C09102=1029.848,308.460,372.432,171.179,46.085,158.925
C09103=1029.841,308.212,372.466,171.174,46.085,158.924
C09104=1029.833,307.965,372.499,171.169,46.086,158.924
C09105=1029.826,307.717,372.532,171.165,46.085,158.923
C09106=1029.819,307.470,372.565,171.160,46.086,158.923
C09107=1029.807,307.057,372.620,171.152,46.086,158.922
C09108=1029.795,306.645,372.676,171.145,46.086,158.921
C09109=1029.784,306.233,372.731,171.136,46.086,158.920
C09110=1029.772,305.821,372.786,171.128,46.087,158.919
C09111=1029.765,305.573,372.819,171.124,46.087,158.919
C09112=1029.758,305.326,372.853,171.119,46.087,158.918
C09113=1029.751,305.077,372.886,171.115,46.087,158.918
C09114=1029.744,304.831,372.919,171.110,46.087,158.917
C09115=1029.737,304.582,372.952,171.105,46.088,158.917
C09116=1029.731,304.335,372.985,171.100,46.088,158.916
C09117=1029.723,304.087,373.018,171.096,46.088,158.916
C09118=1029.717,303.840,373.051,171.092,46.088,158.915
C09119=1029.709,303.592,373.085,171.087,46.088,158.915
C09120=1029.703,303.344,373.117,171.082,46.089,158.914
C09121=1029.695,303.097,373.150,171.077,46.088,158.914
C09122=1029.689,302.850,373.183,171.073,46.089,158.913
C09123=1029.682,302.601,373.216,171.069,46.089,158.913
C09124=1029.674,302.353,373.249,171.064,46.089,158.912
C09125=1029.668,302.106,373.282,171.060,46.089,158.912
C09126=1029.661,301.859,373.315,171.054,46.090,158.911
C09127=1029.654,301.610,373.348,171.050,46.090,158.911
C09128=1029.647,301.363,373.380,171.045,46.090,158.911
C09129=1029.641,301.115,373.413,171.041,46.090,158.910
C09130=1029.634,300.867,373.446,171.037,46.091,158.910
C09131=1029.626,300.620,373.479,171.033,46.091,158.909
C09132=1029.620,300.372,373.512,171.028,46.091,158.909
C09133=1029.613,300.124,373.545,171.023,46.092,158.908
C09134=1029.606,299.877,373.577,171.018,46.092,158.908
C09135=1029.600,299.629,373.610,171.014,46.092,158.907
C09136=1029.593,299.381,373.643,171.009,46.092,158.907
C09137=1029.586,299.134,373.675,171.005,46.093,158.906
C09138=1029.579,298.885,373.708,171.001,46.093,158.906
C09139=1029.573,298.638,373.741,170.996,46.093,158.906
C09140=1029.566,298.390,373.774,170.992,46.094,158.905
C09141=1029.559,298.142,373.806,170.988,46.094,158.905
C09142=1029.552,297.894,373.839,170.983,46.094,158.904
C09143=1029.546,297.647,373.872,170.978,46.094,158.904
C09144=1029.539,297.399,373.904,170.973,46.095,158.903
C09145=1029.532,297.151,373.937,170.969,46.095,158.903
C09146=1029.526,296.904,373.970,170.965,46.096,158.903
C09147=1029.518,296.656,374.002,170.961,46.096,158.902
C09148=1029.512,296.408,374.035,170.956,46.096,158.902
C09149=1029.506,296.161,374.068,170.952,46.097,158.901
C09150=1029.499,295.913,374.100,170.948,46.097,158.901
C09151=1029.492,295.665,374.133,170.943,46.097,158.900
C09152=1029.486,295.417,374.166,170.939,46.097,158.900
C09153=1029.479,295.169,374.197,170.934,46.098,158.900
C09154=1029.473,294.922,374.230,170.930,46.098,158.899
C09155=1029.466,294.674,374.263,170.926,46.098,158.899
C09156=1029.459,294.426,374.295,170.921,46.099,158.898
C09157=1029.452,294.179,374.328,170.917,46.099,158.898
C09158=1029.446,293.931,374.360,170.913,46.099,158.897
C09159=1029.439,293.684,374.392,170.909,46.100,158.897
C09160=1029.432,293.435,374.425,170.904,46.101,158.897
C09161=1029.425,293.187,374.456,170.900,46.101,158.896
C09162=1029.418,292.940,374.488,170.895,46.102,158.896
C09163=1029.407,292.544,374.540,170.888,46.103,158.895
C09164=1029.397,292.150,374.591,170.882,46.103,158.895
C09165=1029.385,291.754,374.642,170.874,46.104,158.894
C09166=1029.375,291.359,374.693,170.868,46.105,158.894
C09167=1029.368,291.112,374.725,170.864,46.105,158.893
C09168=1029.361,290.864,374.757,170.860,46.106,158.893
C09169=1029.354,290.616,374.788,170.854,46.107,158.893
C09170=1029.348,290.367,374.821,170.850,46.107,158.892
C09171=1029.341,290.120,374.853,170.846,46.108,158.892
C09172=1029.334,289.872,374.884,170.842,46.109,158.891
C09173=1029.327,289.625,374.916,170.837,46.109,158.891
C09174=1029.320,289.377,374.948,170.833,46.109,158.891
C09175=1029.314,289.129,374.980,170.829,46.110,158.890
C09176=1029.307,288.882,375.012,170.825,46.111,158.890
C09177=1029.300,288.633,375.044,170.820,46.111,158.890
C09178=1029.293,288.385,375.075,170.816,46.112,158.889
C09179=1029.286,288.137,375.107,170.812,46.113,158.889
C09180=1029.279,287.890,375.139,170.808,46.113,158.889
C09181=1029.273,287.642,375.170,170.804,46.114,158.888
C09182=1029.267,287.394,375.202,170.799,46.114,158.888
C09183=1029.260,287.146,375.234,170.795,46.115,158.888
C09184=1029.253,286.899,375.266,170.791,46.116,158.887
C09185=1029.246,286.651,375.297,170.787,46.117,158.887
C09186=1029.239,286.403,375.329,170.783,46.117,158.887
C09187=1029.233,286.155,375.360,170.778,46.117,158.886
C09188=1029.226,285.907,375.392,170.774,46.118,158.886
C09189=1029.219,285.658,375.423,170.770,46.119,158.886
C09190=1029.212,285.410,375.455,170.766,46.120,158.885
C09191=1029.205,285.163,375.486,170.762,46.121,158.885
C09192=1029.198,284.915,375.518,170.757,46.121,158.885
C09193=1029.192,284.667,375.549,170.753,46.122,158.884
C09194=1029.185,284.419,375.581,170.749,46.123,158.884
C09195=1029.178,284.171,375.612,170.745,46.124,158.884
C09196=1029.172,283.923,375.643,170.741,46.124,158.883
C09197=1029.164,283.675,375.674,170.737,46.125,158.883
C09198=1029.157,283.428,375.706,170.733,46.126,158.883
C09199=1029.151,283.180,375.737,170.729,46.126,158.883
C09200=1029.144,282.932,375.769,170.725,46.127,158.882
C09201=1029.137,282.684,375.800,170.721,46.128,158.882
C09202=1029.130,282.436,375.831,170.717,46.128,158.882
C09203=1029.124,282.187,375.862,170.713,46.129,158.881
C09204=1029.117,281.939,375.894,170.709,46.130,158.881
C09205=1029.111,281.692,375.925,170.705,46.131,158.881
C09206=1029.103,281.444,375.956,170.701,46.132,158.881
C09207=1029.097,281.197,375.987,170.696,46.133,158.880
C09208=1029.091,280.948,376.018,170.692,46.133,158.880
C09209=1029.084,280.700,376.049,170.688,46.134,158.880
C09210=1029.077,280.452,376.080,170.684,46.135,158.879
C09211=1029.070,280.205,376.112,170.680,46.136,158.879
C09212=1029.064,279.956,376.143,170.676,46.137,158.879
C09213=1029.057,279.708,376.174,170.672,46.138,158.879
C09214=1029.051,279.460,376.205,170.668,46.139,158.878
C09215=1029.043,279.213,376.236,170.664,46.139,158.878
C09216=1029.037,278.965,376.267,170.660,46.140,158.878
C09217=1029.031,278.717,376.298,170.656,46.141,158.877
C09218=1029.024,278.469,376.330,170.652,46.142,158.877
C09219=1029.014,278.086,376.377,170.646,46.143,158.877
C09220=1029.003,277.703,376.426,170.640,46.144,158.876
C09221=1028.993,277.320,376.473,170.634,46.146,158.876
C09222=1028.983,276.937,376.521,170.628,46.147,158.876
C09223=1028.976,276.689,376.551,170.624,46.148,158.875
C09224=1028.969,276.441,376.582,170.619,46.149,158.875
C09225=1028.963,276.193,376.612,170.615,46.150,158.875
C09226=1028.956,275.946,376.643,170.611,46.151,158.874
C09227=1028.949,275.697,376.674,170.607,46.152,158.874
C09228=1028.942,275.449,376.705,170.603,46.153,158.874
C09229=1028.935,275.201,376.736,170.599,46.154,158.874
C09230=1028.930,274.953,376.766,170.596,46.154,158.874
C09231=1028.923,274.705,376.797,170.592,46.155,158.873
C09232=1028.916,274.457,376.827,170.588,46.156,158.873
C09233=1028.909,274.209,376.859,170.584,46.157,158.873
C09234=1028.902,273.962,376.889,170.580,46.158,158.873
C09235=1028.896,273.713,376.919,170.576,46.159,158.872
C09236=1028.889,273.465,376.951,170.572,46.160,158.872
C09237=1028.882,273.217,376.981,170.568,46.161,158.872
C09238=1028.876,272.969,377.011,170.564,46.162,158.872
C09239=1028.869,272.721,377.041,170.561,46.163,158.871
C09240=1028.862,272.473,377.073,170.557,46.164,158.871
C09241=1028.855,272.225,377.103,170.553,46.165,158.871
C09242=1028.849,271.977,377.133,170.549,46.166,158.871
C09243=1028.842,271.729,377.163,170.545,46.167,158.870
C09244=1028.836,271.480,377.194,170.540,46.168,158.870
C09245=1028.829,271.233,377.225,170.537,46.170,158.870
C09246=1028.823,270.985,377.255,170.534,46.170,158.870
C09247=1028.816,270.736,377.286,170.530,46.172,158.870
C09248=1028.810,270.489,377.316,170.526,46.173,158.870
C09249=1028.803,270.240,377.347,170.522,46.174,158.869
C09250=1028.796,269.992,377.377,170.518,46.175,158.869
C09251=1028.789,269.744,377.406,170.513,46.176,158.869
C09252=1028.783,269.496,377.437,170.511,46.177,158.869
C09253=1028.776,269.248,377.467,170.507,46.178,158.869
C09254=1028.769,269.000,377.497,170.503,46.179,158.868
C09255=1028.763,268.752,377.528,170.499,46.180,158.868
C09256=1028.756,268.504,377.558,170.495,46.181,158.868
C09257=1028.750,268.256,377.588,170.491,46.183,158.868
C09258=1028.743,268.007,377.618,170.487,46.184,158.867
C09259=1028.736,267.760,377.648,170.484,46.184,158.867
C09260=1028.730,267.511,377.679,170.480,46.185,158.867
C09261=1028.723,267.263,377.709,170.476,46.187,158.867
C09262=1028.716,267.016,377.739,170.472,46.188,158.867
C09263=1028.710,266.767,377.769,170.468,46.189,158.867
C09264=1028.703,266.520,377.799,170.465,46.190,158.867
C09265=1028.696,266.271,377.829,170.461,46.191,158.866
C09266=1028.689,266.023,377.860,170.457,46.192,158.866
C09267=1028.683,265.775,377.889,170.453,46.194,158.866
C09268=1028.676,265.527,377.919,170.449,46.195,158.866
C09269=1028.670,265.279,377.949,170.445,46.196,158.865
C09270=1028.662,265.031,377.979,170.442,46.197,158.865
C09271=1028.657,264.782,378.009,170.438,46.198,158.865
C09272=1028.650,264.534,378.039,170.434,46.199,158.865
C09273=1028.643,264.286,378.069,170.431,46.201,158.865
C09274=1028.636,264.039,378.099,170.427,46.202,158.865
C09275=1028.626,263.660,378.144,170.422,46.204,158.865
C09276=1028.616,263.282,378.189,170.416,46.205,158.864
C09277=1028.606,262.904,378.235,170.410,46.208,158.864
C09278=1028.595,262.525,378.280,170.404,46.210,158.864
C09279=1028.590,262.277,378.311,170.400,46.211,158.864
C09280=1028.583,262.029,378.340,170.397,46.212,158.864
C09281=1028.576,261.781,378.370,170.393,46.213,158.863
C09282=1028.569,261.532,378.399,170.390,46.215,158.863
C09283=1028.563,261.285,378.429,170.385,46.216,158.863
C09284=1028.557,261.037,378.460,170.382,46.217,158.863
C09285=1028.549,260.788,378.488,170.379,46.218,158.863
C09286=1028.543,260.541,378.518,170.375,46.220,158.863
C09287=1028.536,260.292,378.547,170.371,46.221,158.862
C09288=1028.530,260.044,378.577,170.367,46.223,158.862
C09289=1028.523,259.796,378.607,170.363,46.224,158.862
C09290=1028.516,259.548,378.635,170.360,46.225,158.862
C09291=1028.509,259.299,378.665,170.357,46.227,158.862
C09292=1028.502,259.052,378.694,170.353,46.228,158.862
C09293=1028.495,258.803,378.724,170.349,46.229,158.862
C09294=1028.489,258.555,378.753,170.345,46.231,158.862
C09295=1028.481,258.307,378.782,170.341,46.233,158.861
C09296=1028.475,258.059,378.811,170.339,46.234,158.861
C09297=1028.468,257.810,378.841,170.334,46.235,158.861
C09298=1028.462,257.562,378.870,170.331,46.237,158.861
C09299=1028.455,257.314,378.899,170.327,46.238,158.861
C09300=1028.448,257.066,378.928,170.323,46.239,158.861
C09301=1028.441,256.817,378.957,170.320,46.241,158.861
C09302=1028.434,256.569,378.987,170.316,46.242,158.861
C09303=1028.428,256.321,379.016,170.313,46.244,158.861
C09304=1028.422,256.073,379.046,170.309,46.245,158.860
C09305=1028.414,255.824,379.074,170.306,46.246,158.860
C09306=1028.408,255.576,379.103,170.302,46.248,158.860
C09307=1028.401,255.328,379.134,170.298,46.250,158.860
C09308=1028.395,255.080,379.163,170.294,46.251,158.860
C09309=1028.388,254.832,379.191,170.291,46.252,158.860
C09310=1028.381,254.583,379.220,170.288,46.254,158.860
C09311=1028.375,254.335,379.249,170.284,46.255,158.860
C09312=1028.368,254.087,379.278,170.280,46.257,158.860
C09313=1028.361,253.838,379.308,170.276,46.258,158.860
C09314=1028.354,253.591,379.337,170.273,46.259,158.860
C09315=1028.348,253.343,379.366,170.270,46.261,158.859
C09316=1028.341,253.094,379.395,170.266,46.263,158.859
C09317=1028.335,252.846,379.425,170.262,46.264,158.859
C09318=1028.328,252.598,379.453,170.259,46.266,158.859
C09319=1028.322,252.350,379.482,170.255,46.267,158.859
C09320=1028.315,252.101,379.511,170.252,46.268,158.859
C09321=1028.308,251.853,379.540,170.249,46.270,158.859
C09322=1028.302,251.605,379.570,170.245,46.271,158.859
C09323=1028.295,251.356,379.598,170.241,46.273,158.859
C09324=1028.288,251.108,379.627,170.238,46.275,158.859
C09325=1028.282,250.860,379.656,170.235,46.275,158.859
C09326=1028.276,250.612,379.685,170.231,46.277,158.858
C09327=1028.269,250.364,379.714,170.227,46.279,158.858
C09328=1028.262,250.115,379.743,170.224,46.280,158.858
C09329=1028.256,249.867,379.772,170.221,46.282,158.858
C09330=1028.250,249.619,379.801,170.217,46.283,158.858
C09331=1028.239,249.239,379.846,170.211,46.286,158.858
C09332=1028.229,248.860,379.890,170.206,46.288,158.858
C09333=1028.220,248.480,379.933,170.201,46.290,158.858
C09334=1028.210,248.100,379.978,170.196,46.292,158.858
C09335=1028.203,247.852,380.007,170.192,46.294,158.858
C09336=1028.196,247.604,380.035,170.188,46.296,158.858
C09337=1028.190,247.356,380.064,170.186,46.297,158.858
C09338=1028.184,247.107,380.093,170.182,46.299,158.857
C09339=1028.178,246.859,380.122,170.178,46.300,158.857
C09340=1028.170,246.610,380.150,170.175,46.302,158.857
C09341=1028.164,246.362,380.179,170.172,46.303,158.857
C09342=1028.158,246.114,380.208,170.168,46.305,158.857
C09343=1028.151,245.866,380.237,170.165,46.306,158.857
C09344=1028.145,245.617,380.265,170.161,46.308,158.857
C09345=1028.139,245.369,380.294,170.158,46.310,158.857
C09346=1028.132,245.121,380.323,170.155,46.311,158.857
C09347=1028.126,244.873,380.352,170.151,46.313,158.857
C09348=1028.119,244.624,380.380,170.147,46.314,158.857
C09349=1028.113,244.376,380.409,170.145,46.316,158.857
C09350=1028.106,244.128,380.438,170.141,46.317,158.857
C09351=1028.100,243.879,380.466,170.137,46.319,158.857
C09352=1028.093,243.631,380.495,170.134,46.320,158.857
C09353=1028.087,243.383,380.523,170.131,46.322,158.857
C09354=1028.080,243.134,380.552,170.127,46.324,158.856
C09355=1028.073,242.887,380.580,170.124,46.326,158.857
C09356=1028.067,242.638,380.609,170.121,46.327,158.857
C09357=1028.061,242.390,380.637,170.117,46.329,158.856
C09358=1028.055,242.141,380.666,170.114,46.331,158.856
C09359=1028.048,241.893,380.694,170.110,46.332,158.856
C09360=1028.042,241.645,380.722,170.107,46.334,158.856
C09361=1028.035,241.397,380.751,170.104,46.336,158.856
C09362=1028.029,241.148,380.779,170.100,46.338,158.856
C09363=1028.022,240.900,380.808,170.097,46.339,158.856
C09364=1028.014,240.651,380.836,170.094,46.341,158.856
C09365=1028.008,240.403,380.865,170.090,46.342,158.856
C09366=1028.002,240.155,380.892,170.086,46.344,158.856
C09367=1027.996,239.906,380.921,170.084,46.346,158.856
C09368=1027.989,239.658,380.949,170.080,46.348,158.856
C09369=1027.982,239.410,380.977,170.076,46.349,158.856
C09370=1027.975,239.161,381.005,170.074,46.351,158.856
C09371=1027.969,238.913,381.034,170.070,46.353,158.856
C09372=1027.962,238.665,381.061,170.066,46.355,158.856
C09373=1027.956,238.416,381.089,170.064,46.357,158.856
C09374=1027.949,238.168,381.117,170.060,46.358,158.856
C09375=1027.942,237.920,381.145,170.056,46.360,158.856
C09376=1027.936,237.671,381.174,170.054,46.362,158.856
C09377=1027.929,237.423,381.201,170.050,46.364,158.856
C09378=1027.923,237.174,381.229,170.046,46.365,158.856
C09379=1027.916,236.926,381.258,170.044,46.367,158.856
C09380=1027.909,236.678,381.285,170.040,46.369,158.856
C09381=1027.903,236.429,381.314,170.037,46.371,158.856
C09382=1027.896,236.181,381.341,170.034,46.373,158.856
C09383=1027.890,235.932,381.369,170.030,46.374,158.856
C09384=1027.883,235.684,381.397,170.027,46.377,158.856
C09385=1027.877,235.437,381.425,170.024,46.378,158.856
C09386=1027.870,235.188,381.453,170.020,46.380,158.856
C09387=1027.859,234.802,381.496,170.015,46.383,158.856
C09388=1027.850,234.417,381.539,170.010,46.386,158.856
C09389=1027.839,234.031,381.582,170.005,46.389,158.856
C09390=1027.829,233.645,381.626,170.000,46.392,158.856
C09391=1027.823,233.397,381.653,169.997,46.394,158.856
C09392=1027.816,233.148,381.681,169.993,46.395,158.856
C09393=1027.810,232.900,381.709,169.991,46.397,158.856
C09394=1027.803,232.651,381.737,169.987,46.399,158.856
C09395=1027.797,232.403,381.765,169.983,46.401,158.856
C09396=1027.790,232.154,381.792,169.981,46.403,158.856
C09397=1027.783,231.906,381.820,169.977,46.405,158.857
C09398=1027.777,231.657,381.848,169.973,46.407,158.856
C09399=1027.770,231.410,381.875,169.971,46.409,158.857
C09400=1027.764,231.161,381.903,169.967,46.410,158.856
C09401=1027.758,230.913,381.931,169.965,46.412,158.857
C09402=1027.751,230.664,381.959,169.961,46.414,158.857
C09403=1027.744,230.416,381.987,169.958,46.416,158.857
C09404=1027.738,230.167,382.015,169.955,46.418,158.857
C09405=1027.731,229.918,382.041,169.951,46.420,158.857
C09406=1027.725,229.671,382.068,169.948,46.422,158.857
C09407=1027.718,229.422,382.096,169.945,46.424,158.857
C09408=1027.711,229.174,382.124,169.942,46.426,158.857
C09409=1027.705,228.925,382.152,169.939,46.427,158.857
C09410=1027.698,228.677,382.179,169.935,46.430,158.857
C09411=1027.691,228.428,382.206,169.932,46.432,158.857
C09412=1027.685,228.180,382.234,169.929,46.434,158.857
C09413=1027.679,227.932,382.261,169.926,46.436,158.857
C09414=1027.672,227.683,382.289,169.923,46.438,158.857
C09415=1027.665,227.435,382.317,169.920,46.440,158.857
C09416=1027.660,227.186,382.343,169.916,46.442,158.857
C09417=1027.653,226.938,382.371,169.914,46.444,158.857
C09418=1027.645,226.690,382.398,169.910,46.446,158.857
C09419=1027.639,226.441,382.425,169.906,46.448,158.857
C09420=1027.632,226.192,382.453,169.904,46.450,158.858
C09421=1027.626,225.945,382.480,169.900,46.452,158.858
C09422=1027.619,225.696,382.507,169.898,46.454,158.858
C09423=1027.613,225.447,382.535,169.894,46.456,158.858
C09424=1027.606,225.198,382.562,169.891,46.458,158.858
C09425=1027.600,224.950,382.589,169.888,46.460,158.858
C09426=1027.593,224.703,382.616,169.884,46.462,158.858
C09427=1027.586,224.453,382.643,169.881,46.464,158.858
C09428=1027.580,224.205,382.671,169.879,46.466,158.858
C09429=1027.573,223.956,382.697,169.875,46.469,158.858
C09430=1027.566,223.709,382.725,169.873,46.471,158.858
C09431=1027.560,223.459,382.752,169.869,46.472,158.858
C09432=1027.553,223.211,382.779,169.865,46.475,158.858
C09433=1027.546,222.963,382.807,169.863,46.477,158.858
C09434=1027.540,222.715,382.833,169.859,46.479,158.859
C09435=1027.534,222.466,382.861,169.857,46.481,158.859
C09436=1027.527,222.217,382.888,169.853,46.483,158.859
C09437=1027.520,221.970,382.915,169.850,46.485,158.859
C09438=1027.514,221.721,382.942,169.847,46.487,158.859
C09439=1027.507,221.472,382.969,169.844,46.490,158.859
C09440=1027.501,221.224,382.995,169.841,46.492,158.859
C09441=1027.494,220.975,383.023,169.838,46.493,158.859
C09442=1027.488,220.727,383.050,169.834,46.496,158.859
C09443=1027.477,220.333,383.093,169.830,46.499,158.859
C09444=1027.467,219.940,383.136,169.825,46.502,158.859
C09445=1027.456,219.546,383.179,169.819,46.506,158.859
C09446=1027.447,219.153,383.221,169.815,46.509,158.860
C09447=1027.440,218.904,383.248,169.812,46.511,158.860
C09448=1027.433,218.656,383.275,169.809,46.513,158.860
C09449=1027.427,218.407,383.301,169.806,46.516,158.860
C09450=1027.420,218.159,383.329,169.802,46.518,158.860
C09451=1027.413,217.910,383.355,169.800,46.520,158.860
C09452=1027.407,217.662,383.382,169.796,46.522,158.860
C09453=1027.400,217.413,383.408,169.794,46.524,158.860
C09454=1027.393,217.164,383.435,169.791,46.527,158.861
C09455=1027.387,216.917,383.462,169.787,46.529,158.861
C09456=1027.380,216.668,383.489,169.785,46.531,158.861
C09457=1027.374,216.420,383.515,169.781,46.534,158.861
C09458=1027.367,216.171,383.541,169.779,46.536,158.861
C09459=1027.360,215.922,383.568,169.775,46.538,158.861
C09460=1027.353,215.675,383.595,169.772,46.540,158.861
C09461=1027.347,215.425,383.622,169.769,46.542,158.861
C09462=1027.341,215.177,383.648,169.766,46.545,158.861
C09463=1027.334,214.928,383.675,169.763,46.547,158.862
C09464=1027.327,214.680,383.702,169.760,46.549,158.862
C09465=1027.321,214.432,383.728,169.756,46.551,158.862
C09466=1027.314,214.182,383.755,169.754,46.554,158.862
C09467=1027.308,213.934,383.781,169.751,46.556,158.862
C09468=1027.301,213.686,383.808,169.748,46.558,158.862
C09469=1027.294,213.438,383.834,169.745,46.561,158.862
C09470=1027.288,213.189,383.861,169.742,46.563,158.862
C09471=1027.281,212.940,383.888,169.739,46.565,158.863
C09472=1027.274,212.692,383.914,169.735,46.567,158.863
C09473=1027.268,212.443,383.941,169.733,46.570,158.863
C09474=1027.262,212.195,383.967,169.730,46.572,158.863
C09475=1027.255,211.946,383.994,169.727,46.574,158.863
C09476=1027.249,211.698,384.020,169.724,46.576,158.863
C09477=1027.242,211.449,384.047,169.721,46.578,158.863
C09478=1027.236,211.201,384.073,169.718,46.581,158.863
C09479=1027.229,210.952,384.100,169.715,46.583,158.864
C09480=1027.223,210.704,384.126,169.712,46.586,158.864
C09481=1027.216,210.455,384.153,169.709,46.588,158.864
C09482=1027.209,210.207,384.179,169.706,46.590,158.864
C09483=1027.202,209.958,384.205,169.703,46.592,158.864
C09484=1027.196,209.710,384.232,169.700,46.595,158.864
C09485=1027.189,209.461,384.258,169.697,46.598,158.864
C09486=1027.183,209.213,384.284,169.695,46.600,158.865
C09487=1027.176,208.964,384.310,169.691,46.602,158.865
C09488=1027.170,208.715,384.337,169.689,46.605,158.865
C09489=1027.164,208.467,384.363,169.685,46.607,158.865
C09490=1027.157,208.218,384.389,169.682,46.609,158.865
C09491=1027.150,207.970,384.415,169.679,46.611,158.865
C09492=1027.143,207.722,384.442,169.676,46.614,158.865
C09493=1027.137,207.473,384.467,169.674,46.616,158.866
C09494=1027.130,207.224,384.494,169.670,46.619,158.866
C09495=1027.124,206.976,384.520,169.668,46.621,158.866
C09496=1027.117,206.727,384.546,169.665,46.624,158.866
C09497=1027.110,206.479,384.572,169.661,46.626,158.866
C09498=1027.103,206.230,384.598,169.659,46.628,158.866
C09499=1027.093,205.841,384.640,169.654,46.632,158.867
C09500=1027.083,205.452,384.680,169.650,46.636,158.867
C09501=1027.072,205.063,384.720,169.645,46.640,158.867
C09502=1027.062,204.674,384.761,169.640,46.644,158.867
C09503=1027.037,203.632,384.864,169.257,46.541,158.800
C09504=1027.032,203.384,384.888,169.252,46.544,158.800
C09505=1027.025,203.135,384.914,169.249,46.547,158.800
C09506=1027.020,202.887,384.938,169.245,46.551,158.800
C09507=1027.014,202.637,384.963,169.241,46.554,158.801
C09508=1027.008,202.390,384.987,169.237,46.557,158.801
C09509=1027.002,202.140,385.012,169.234,46.561,158.801
C09510=1026.997,201.892,385.036,169.229,46.564,158.801
C09511=1026.991,201.642,385.060,169.225,46.567,158.801
C09512=1026.985,201.394,385.085,169.222,46.570,158.802
C09513=1026.978,201.145,385.109,169.218,46.573,158.802
C09514=1026.973,200.897,385.134,169.214,46.577,158.802
C09515=1026.967,200.648,385.158,169.209,46.580,158.802
C09516=1026.962,200.399,385.183,169.206,46.583,158.803
C09517=1026.956,200.150,385.207,169.202,46.587,158.803
C09518=1026.950,199.902,385.232,169.198,46.590,158.803
C09519=1026.944,199.653,385.256,169.195,46.593,158.803
C09520=1026.938,199.405,385.280,169.191,46.597,158.804
C09521=1026.931,199.156,385.304,169.187,46.600,158.804
C09522=1026.926,198.907,385.328,169.182,46.603,158.804
C09523=1026.919,198.658,385.352,169.179,46.607,158.804
C09524=1026.914,198.409,385.376,169.175,46.610,158.804
C09525=1026.907,198.160,385.400,169.171,46.614,158.805
C09526=1026.902,197.912,385.425,169.167,46.617,158.805
C09527=1026.896,197.662,385.448,169.164,46.620,158.805
C09528=1026.890,197.414,385.472,169.160,46.624,158.805
C09529=1026.884,197.165,385.496,169.156,46.628,158.806
C09530=1026.878,196.916,385.520,169.152,46.631,158.806
C09531=1026.872,196.668,385.544,169.148,46.634,158.806
C09532=1026.866,196.419,385.568,169.145,46.638,158.806
C09533=1026.860,196.170,385.592,169.140,46.641,158.806
C09534=1026.854,195.921,385.616,169.137,46.644,158.807
C09535=1026.848,195.673,385.641,169.133,46.648,158.807
C09536=1026.843,195.424,385.664,169.129,46.651,158.807
C09537=1026.836,195.175,385.688,169.126,46.655,158.808
C09538=1026.831,194.926,385.712,169.122,46.658,158.808
C09539=1026.824,194.677,385.736,169.118,46.661,158.808
C09540=1026.819,194.429,385.760,169.115,46.665,158.808
C09541=1026.813,194.180,385.784,169.111,46.668,158.809
C09542=1026.807,193.930,385.808,169.107,46.672,158.809
C09543=1026.801,193.682,385.831,169.103,46.675,158.809
C09544=1026.795,193.434,385.855,169.099,46.678,158.809
C09545=1026.789,193.185,385.880,169.095,46.682,158.810
C09546=1026.784,192.936,385.903,169.092,46.685,158.810
C09547=1026.778,192.687,385.927,169.088,46.689,158.810
C09548=1026.772,192.438,385.951,169.084,46.693,158.810
C09549=1026.766,192.190,385.975,169.081,46.696,158.810
C09550=1026.761,191.941,385.998,169.077,46.699,158.811
C09551=1026.754,191.692,386.022,169.073,46.703,158.811
C09552=1026.749,191.443,386.046,169.070,46.706,158.811
C09553=1026.743,191.194,386.069,169.066,46.710,158.812
C09554=1026.738,190.946,386.094,169.062,46.713,158.812
C09555=1026.731,190.697,386.118,169.058,46.717,158.812
C09556=1026.725,190.448,386.141,169.054,46.720,158.812
C09557=1026.720,190.199,386.165,169.051,46.723,158.813
C09558=1026.714,189.951,386.189,169.047,46.727,158.813
C09559=1026.708,189.701,386.212,169.044,46.730,158.813
C09560=1026.702,189.453,386.236,169.040,46.734,158.813
C09561=1026.697,189.204,386.259,169.037,46.737,158.814
C09562=1026.691,188.955,386.283,169.033,46.741,158.814
C09563=1026.685,188.707,386.307,169.029,46.744,158.814
C09564=1026.679,188.423,386.334,169.025,46.748,158.814
C09565=1026.672,188.140,386.361,169.021,46.752,158.815
C09566=1026.666,187.858,386.388,169.017,46.756,158.815
C09567=1026.659,187.575,386.415,169.013,46.760,158.815
C09568=1026.653,187.326,386.438,169.009,46.763,158.816
C09569=1026.648,187.078,386.462,169.006,46.767,158.816
C09570=1026.642,186.829,386.485,169.002,46.770,158.816
C09571=1026.637,186.580,386.509,168.999,46.773,158.816
C09572=1026.631,186.331,386.532,168.995,46.777,158.817
C09573=1026.624,186.082,386.556,168.991,46.781,158.817
C09574=1026.619,185.833,386.580,168.988,46.784,158.817
C09575=1026.613,185.585,386.603,168.984,46.788,158.817
C09576=1026.608,185.336,386.626,168.980,46.791,158.818
C09577=1026.603,185.087,386.650,168.977,46.795,158.818
C09578=1026.597,184.838,386.674,168.973,46.798,158.818
C09579=1026.592,184.589,386.697,168.969,46.801,158.818
C09580=1026.586,184.341,386.721,168.966,46.805,158.819
C09581=1026.580,184.092,386.744,168.962,46.808,158.819
C09582=1026.574,183.842,386.768,168.959,46.812,158.819
C09583=1026.568,183.594,386.791,168.956,46.815,158.820
C09584=1026.563,183.345,386.815,168.952,46.818,158.820
C09585=1026.557,183.096,386.838,168.949,46.822,158.820
C09586=1026.551,182.847,386.861,168.945,46.825,158.820
C09587=1026.546,182.598,386.885,168.942,46.828,158.821
C09588=1026.540,182.350,386.907,168.938,46.832,158.821
C09589=1026.534,182.101,386.930,168.934,46.836,158.821
C09590=1026.528,181.851,386.954,168.931,46.840,158.822
C09591=1026.522,181.602,386.977,168.927,46.844,158.822
C09592=1026.516,181.353,386.999,168.924,46.847,158.822
C09593=1026.510,181.105,387.022,168.920,46.851,158.823
C09594=1026.504,180.856,387.045,168.917,46.855,158.823
C09595=1026.498,180.608,387.068,168.913,46.859,158.823
C09596=1026.492,180.359,387.091,168.909,46.863,158.824
C09597=1026.486,180.110,387.114,168.906,46.866,158.824
C09598=1026.480,179.860,387.137,168.902,46.870,158.824
C09599=1026.474,179.612,387.160,168.899,46.873,158.825
C09600=1026.468,179.363,387.183,168.895,46.877,158.825
C09601=1026.462,179.114,387.205,168.893,46.881,158.825
C09602=1026.456,178.865,387.227,168.888,46.884,158.825
C09603=1026.451,178.616,387.250,168.885,46.888,158.826
C09604=1026.445,178.367,387.273,168.882,46.892,158.826
C09605=1026.438,178.118,387.296,168.879,46.895,158.827
C09606=1026.433,177.869,387.319,168.875,46.899,158.827
C09607=1026.427,177.620,387.342,168.872,46.903,158.827
C09608=1026.421,177.371,387.365,168.868,46.906,158.827
C09609=1026.415,177.123,387.387,168.864,46.910,158.828
C09610=1026.409,176.874,387.410,168.861,46.914,158.828
C09611=1026.403,176.625,387.433,168.857,46.918,158.828
C09612=1026.398,176.376,387.456,168.854,46.922,158.829
C09613=1026.391,176.128,387.478,168.850,46.925,158.829
C09614=1026.386,175.878,387.500,168.847,46.929,158.829
C09615=1026.380,175.629,387.523,168.844,46.932,158.830
C09616=1026.374,175.380,387.546,168.840,46.936,158.830
C09617=1026.368,175.132,387.569,168.837,46.940,158.830
C09618=1026.362,174.883,387.592,168.833,46.944,158.831
C09619=1026.356,174.634,387.614,168.830,46.947,158.831
C09620=1026.351,174.384,387.637,168.826,46.951,158.831
C09621=1026.344,174.136,387.659,168.823,46.955,158.832
C09622=1026.339,173.887,387.682,168.819,46.959,158.832
C09623=1026.333,173.638,387.705,168.817,46.962,158.832
C09624=1026.327,173.389,387.727,168.813,46.966,158.833
C09625=1026.321,173.140,387.750,168.810,46.970,158.833
C09626=1026.315,172.891,387.772,168.806,46.973,158.833
C09627=1026.310,172.643,387.795,168.803,46.977,158.834
C09628=1026.304,172.359,387.820,168.799,46.982,158.834
C09629=1026.297,172.076,387.846,168.795,46.986,158.834
C09630=1026.290,171.793,387.872,168.791,46.990,158.835
C09631=1026.284,171.509,387.897,168.788,46.994,158.835
C09632=1026.278,171.261,387.920,168.784,46.998,158.836
C09633=1026.272,171.012,387.943,168.781,47.001,158.836
C09634=1026.266,170.762,387.965,168.778,47.005,158.836
C09635=1026.260,170.514,387.988,168.774,47.009,158.836
C09636=1026.255,170.265,388.011,168.771,47.013,158.837
C09637=1026.249,170.016,388.032,168.767,47.017,158.837
C09638=1026.243,169.767,388.055,168.764,47.020,158.838
C09639=1026.238,169.518,388.077,168.761,47.024,158.838
C09640=1026.232,169.269,388.100,168.757,47.027,158.838
C09641=1026.226,169.020,388.122,168.754,47.031,158.838
C09642=1026.220,168.771,388.145,168.751,47.035,158.839
C09643=1026.215,168.523,388.167,168.747,47.039,158.839
C09644=1026.209,168.274,388.189,168.745,47.042,158.840
C09645=1026.203,168.024,388.212,168.741,47.046,158.840
C09646=1026.197,167.776,388.235,168.737,47.049,158.840
C09647=1026.192,167.526,388.257,168.735,47.053,158.840
C09648=1026.186,167.278,388.279,168.731,47.057,158.841
C09649=1026.181,167.029,388.301,168.728,47.061,158.841
C09650=1026.175,166.780,388.324,168.725,47.065,158.842
C09651=1026.169,166.531,388.346,168.721,47.069,158.842
C09652=1026.164,166.282,388.368,168.718,47.072,158.842
C09653=1026.158,166.033,388.390,168.715,47.075,158.842
C09654=1026.152,165.784,388.413,168.711,47.079,158.843
C09655=1026.146,165.535,388.435,168.708,47.083,158.843
C09656=1026.141,165.287,388.458,168.705,47.087,158.844
C09657=1026.136,165.037,388.480,168.701,47.091,158.844
C09658=1026.129,164.788,388.502,168.699,47.094,158.844
C09659=1026.124,164.539,388.524,168.696,47.098,158.845
C09660=1026.119,164.291,388.547,168.692,47.101,158.845
C09661=1026.113,164.042,388.569,168.689,47.105,158.845
C09662=1026.107,163.793,388.592,168.686,47.109,158.846
C09663=1026.102,163.544,388.613,168.683,47.113,158.846
C09664=1026.096,163.295,388.635,168.679,47.117,158.846
C09665=1026.090,163.046,388.658,168.676,47.120,158.847
C09666=1026.085,162.796,388.680,168.673,47.124,158.847
C09667=1026.079,162.548,388.702,168.669,47.127,158.847
C09668=1026.073,162.299,388.725,168.666,47.131,158.847
C09669=1026.068,162.049,388.747,168.663,47.135,158.848
C09670=1026.062,161.801,388.769,168.660,47.139,158.848
C09671=1026.057,161.552,388.791,168.657,47.143,158.849
C09672=1026.052,161.303,388.813,168.654,47.146,158.849
C09673=1026.046,161.054,388.836,168.651,47.150,158.849
C09674=1026.040,160.805,388.857,168.648,47.153,158.850
C09675=1026.035,160.556,388.879,168.644,47.157,158.850
C09676=1026.029,160.307,388.902,168.641,47.161,158.850
C09677=1026.023,160.058,388.924,168.638,47.165,158.851
C09678=1026.019,159.809,388.946,168.635,47.168,158.851
C09679=1026.013,159.560,388.969,168.631,47.172,158.851
C09680=1026.007,159.312,388.990,168.628,47.176,158.852
C09681=1026.002,159.062,389.012,168.625,47.180,158.852
C09682=1025.996,158.813,389.034,168.623,47.183,158.852
C09683=1025.990,158.565,389.055,168.619,47.187,158.853
C09684=1025.984,158.315,389.077,168.616,47.191,158.853
C09685=1025.978,158.066,389.099,168.613,47.195,158.854
C09686=1025.973,157.817,389.120,168.609,47.199,158.854
C09687=1025.967,157.568,389.142,168.606,47.203,158.854
C09688=1025.961,157.319,389.163,168.603,47.206,158.855
C09689=1025.955,157.070,389.185,168.599,47.210,158.855
C09690=1025.949,156.822,389.208,168.597,47.214,158.855
C09691=1025.943,156.572,389.229,168.594,47.218,158.856
C09692=1025.935,156.207,389.261,168.588,47.224,158.856
C09693=1025.927,155.843,389.292,168.584,47.229,158.857
C09694=1025.918,155.478,389.324,168.580,47.235,158.857
C09695=1025.910,155.113,389.356,168.575,47.241,158.858
C09696=1025.904,154.865,389.377,168.572,47.245,158.858
C09697=1025.899,154.615,389.399,168.569,47.249,158.859
C09698=1025.892,154.366,389.421,168.566,47.253,158.859
C09699=1025.887,154.117,389.442,168.563,47.256,158.859
C09700=1025.881,153.868,389.464,168.559,47.260,158.860
C09701=1025.876,153.619,389.485,168.557,47.264,158.860
C09702=1025.870,153.370,389.506,168.554,47.268,158.861
C09703=1025.864,153.121,389.528,168.551,47.272,158.861
C09704=1025.858,152.872,389.549,168.547,47.276,158.861
C09705=1025.852,152.623,389.571,168.544,47.279,158.862
C09706=1025.847,152.374,389.592,168.541,47.284,158.862
C09707=1025.840,152.125,389.614,168.538,47.288,158.862
C09708=1025.835,151.876,389.634,168.535,47.292,158.863
C09709=1025.829,151.627,389.656,168.532,47.295,158.863
C09710=1025.823,151.378,389.677,168.529,47.299,158.864
C09711=1025.817,151.129,389.699,168.525,47.303,158.864
C09712=1025.812,150.880,389.720,168.523,47.307,158.864
C09713=1025.807,150.630,389.742,168.520,47.311,158.865
C09714=1025.801,150.382,389.763,168.517,47.315,158.865
C09715=1025.795,150.133,389.785,168.513,47.319,158.866
C09716=1025.789,149.884,389.806,168.510,47.323,158.866
C09717=1025.783,149.634,389.827,168.507,47.327,158.866
C09718=1025.778,149.386,389.848,168.504,47.330,158.867
C09719=1025.772,149.136,389.870,168.502,47.335,158.867
C09720=1025.766,148.888,389.891,168.498,47.339,158.868
C09721=1025.760,148.638,389.912,168.495,47.342,158.868
C09722=1025.755,148.390,389.933,168.492,47.346,158.868
C09723=1025.749,148.140,389.955,168.489,47.350,158.869
C09724=1025.743,147.891,389.975,168.485,47.354,158.869
C09725=1025.737,147.642,389.997,168.483,47.358,158.869
C09726=1025.732,147.394,390.018,168.480,47.362,158.870
C09727=1025.726,147.144,390.039,168.477,47.366,158.870
C09728=1025.720,146.895,390.060,168.474,47.370,158.871
C09729=1025.715,146.647,390.082,168.470,47.374,158.871
C09730=1025.709,146.397,390.103,168.468,47.377,158.871
C09731=1025.703,146.148,390.124,168.465,47.382,158.872
C09732=1025.697,145.899,390.145,168.462,47.386,158.872
C09733=1025.691,145.650,390.165,168.458,47.390,158.873
C09734=1025.685,145.401,390.186,168.455,47.393,158.873
C09735=1025.680,145.152,390.208,168.453,47.398,158.873
C09736=1025.674,144.903,390.228,168.450,47.402,158.874
C09737=1025.668,144.654,390.250,168.447,47.405,158.874
C09738=1025.662,144.405,390.270,168.443,47.409,158.874
C09739=1025.656,144.156,390.291,168.441,47.414,158.875
C09740=1025.647,143.739,390.326,168.436,47.420,158.876
C09741=1025.637,143.322,390.362,168.431,47.427,158.876
C09742=1025.627,142.905,390.396,168.426,47.434,158.877
C09743=1025.618,142.488,390.431,168.421,47.440,158.878
C09744=1025.611,142.239,390.452,168.418,47.445,158.878
C09745=1025.606,141.990,390.473,168.415,47.448,158.879
C09746=1025.601,141.741,390.494,168.412,47.452,158.879
C09747=1025.595,141.491,390.515,168.409,47.456,158.879
C09748=1025.589,141.243,390.535,168.406,47.461,158.880
C09749=1025.583,140.994,390.556,168.403,47.464,158.880
C09750=1025.577,140.744,390.577,168.400,47.468,158.881
C09751=1025.572,140.496,390.598,168.397,47.472,158.881
C09752=1025.565,140.211,390.622,168.394,47.477,158.881
C09753=1025.559,139.927,390.646,168.390,47.481,158.882
C09754=1025.553,139.644,390.669,168.387,47.486,158.882
C09755=1025.546,139.360,390.693,168.383,47.491,158.883
C09756=1025.540,139.111,390.713,168.380,47.495,158.883
C09757=1025.534,138.861,390.734,168.378,47.498,158.884
C09758=1025.528,138.613,390.756,168.375,47.502,158.884
C09759=1025.523,138.363,390.776,168.372,47.507,158.884
C09760=1025.517,138.114,390.796,168.369,47.510,158.885
C09761=1025.511,137.865,390.817,168.365,47.514,158.885
C09762=1025.505,137.616,390.837,168.363,47.519,158.886
C09763=1025.499,137.367,390.859,168.360,47.523,158.886
C09764=1025.494,137.118,390.879,168.357,47.526,158.886
C09765=1025.488,136.869,390.899,168.354,47.530,158.887
C09766=1025.483,136.620,390.920,168.352,47.535,158.887
C09767=1025.476,136.370,390.940,168.348,47.539,158.888
C09768=1025.471,136.122,390.961,168.345,47.542,158.888
C09769=1025.465,135.873,390.982,168.343,47.547,158.889
C09770=1025.459,135.623,391.002,168.340,47.551,158.889
C09771=1025.453,135.374,391.023,168.337,47.554,158.889
C09772=1025.447,135.125,391.043,168.334,47.559,158.890
C09773=1025.442,134.876,391.063,168.331,47.563,158.890
C09774=1025.436,134.626,391.084,168.328,47.567,158.891
C09775=1025.430,134.377,391.104,168.325,47.571,158.891
C09776=1025.424,134.129,391.125,168.322,47.575,158.891
C09777=1025.419,133.880,391.145,168.320,47.579,158.892
C09778=1025.412,133.630,391.166,168.317,47.583,158.892
C09779=1025.407,133.381,391.186,168.314,47.587,158.893
C09780=1025.401,133.133,391.206,168.311,47.592,158.893
C09781=1025.396,132.883,391.227,168.308,47.595,158.894
C09782=1025.389,132.634,391.247,168.305,47.599,158.894
C09783=1025.384,132.385,391.268,168.302,47.604,158.894
C09784=1025.378,132.136,391.288,168.299,47.607,158.895
C09785=1025.373,131.887,391.308,168.297,47.611,158.895
C09786=1025.367,131.638,391.328,168.294,47.615,158.896
C09787=1025.361,131.388,391.349,168.291,47.619,158.896
C09788=1025.355,131.139,391.369,168.287,47.624,158.896
C09789=1025.349,130.890,391.389,168.285,47.627,158.897
C09790=1025.343,130.641,391.409,168.282,47.632,158.897
C09791=1025.338,130.392,391.430,168.279,47.636,158.898
C09792=1025.332,130.143,391.450,168.276,47.639,158.898
C09793=1025.326,129.894,391.471,168.274,47.644,158.899
C09794=1025.320,129.645,391.491,168.271,47.648,158.899
C09795=1025.315,129.395,391.510,168.267,47.652,158.899
C09796=1025.309,129.147,391.530,168.265,47.656,158.900
C09797=1025.302,128.897,391.550,168.262,47.661,158.900
C09798=1025.296,128.648,391.570,168.259,47.664,158.901
C09799=1025.291,128.399,391.591,168.257,47.669,158.901
C09800=1025.285,128.150,391.610,168.254,47.673,158.902
C09801=1025.279,127.901,391.630,168.250,47.677,158.902
C09802=1025.273,127.652,391.650,168.247,47.681,158.902
C09803=1025.267,127.403,391.670,168.245,47.686,158.903
C09804=1025.261,127.154,391.691,168.242,47.689,158.903
C09805=1025.256,126.904,391.710,168.240,47.694,158.904
C09806=1025.250,126.655,391.730,168.237,47.698,158.904
C09807=1025.244,126.406,391.750,168.233,47.702,158.905
C09808=1025.238,126.158,391.770,168.230,47.706,158.905
C09809=1025.231,125.907,391.790,168.228,47.711,158.906
C09810=1025.226,125.658,391.810,168.225,47.715,158.906
C09811=1025.220,125.410,391.830,168.222,47.719,158.907
C09812=1025.214,125.160,391.849,168.220,47.723,158.907
C09813=1025.208,124.911,391.869,168.217,47.727,158.907
C09814=1025.202,124.663,391.889,168.213,47.731,158.908
C09815=1025.197,124.413,391.909,168.210,47.735,158.908
C09816=1025.190,124.128,391.932,168.208,47.740,158.909
C09817=1025.184,123.845,391.954,168.205,47.745,158.909
C09818=1025.177,123.560,391.977,168.201,47.750,158.910
C09819=1025.170,123.277,391.999,168.199,47.754,158.910
C09820=1025.165,123.028,392.020,168.195,47.758,158.911
C09821=1025.159,122.779,392.040,168.192,47.763,158.911
C09822=1025.153,122.529,392.059,168.189,47.767,158.912
C09823=1025.147,122.280,392.079,168.187,47.770,158.912
C09824=1025.141,122.031,392.099,168.184,47.775,158.912
C09825=1025.135,121.782,392.118,168.181,47.779,158.913
C09826=1025.129,121.533,392.138,168.179,47.783,158.913
C09827=1025.124,121.283,392.158,168.176,47.787,158.914
C09828=1025.118,121.034,392.178,168.173,47.792,158.914
C09829=1025.112,120.785,392.198,168.171,47.795,158.915
C09830=1025.106,120.536,392.217,168.168,47.799,158.915
C09831=1025.100,120.287,392.237,168.164,47.804,158.915
C09832=1025.095,120.038,392.257,168.161,47.808,158.916
C09833=1025.089,119.789,392.277,168.159,47.812,158.916
C09834=1025.084,119.539,392.296,168.156,47.816,158.917
C09835=1025.078,119.290,392.316,168.153,47.820,158.917
C09836=1025.072,119.041,392.336,168.151,47.824,158.918
C09837=1025.066,118.792,392.356,168.148,47.828,158.918
C09838=1025.060,118.543,392.375,168.145,47.833,158.919
C09839=1025.054,118.294,392.395,168.142,47.836,158.919
C09840=1025.049,118.044,392.415,168.140,47.840,158.919
C09841=1025.043,117.795,392.435,168.137,47.845,158.920
C09842=1025.038,117.546,392.454,168.134,47.849,158.920
C09843=1025.032,117.297,392.474,168.132,47.853,158.921
C09844=1025.026,117.048,392.493,168.129,47.857,158.921
C09845=1025.020,116.799,392.513,168.126,47.861,158.921
C09846=1025.014,116.549,392.532,168.124,47.865,158.922
C09847=1025.008,116.301,392.552,168.121,47.869,158.922
C09848=1025.003,116.051,392.572,168.118,47.873,158.923
C09849=1024.997,115.802,392.592,168.115,47.877,158.923
C09850=1024.992,115.553,392.611,168.113,47.881,158.924
C09851=1024.986,115.304,392.631,168.110,47.886,158.924
C09852=1024.980,115.054,392.650,168.107,47.889,158.925
C09853=1024.974,114.805,392.670,168.105,47.893,158.925
C09854=1024.969,114.557,392.689,168.102,47.898,158.925
C09855=1024.964,114.307,392.709,168.099,47.902,158.926
C09856=1024.958,114.058,392.729,168.096,47.905,158.926
C09857=1024.952,113.809,392.748,168.094,47.910,158.927
C09858=1024.947,113.559,392.768,168.091,47.914,158.927
C09859=1024.941,113.311,392.788,168.088,47.918,158.927
C09860=1024.935,113.061,392.807,168.086,47.922,158.928
C09861=1024.929,112.812,392.826,168.083,47.926,158.928
C09862=1024.923,112.563,392.846,168.080,47.930,158.929
C09863=1024.918,112.313,392.865,168.077,47.934,158.929
C09864=1024.912,112.064,392.884,168.074,47.938,158.930
C09865=1024.906,111.815,392.904,168.071,47.943,158.930
C09866=1024.900,111.566,392.924,168.068,47.947,158.930
C09867=1024.895,111.317,392.943,168.066,47.951,158.931
C09868=1024.889,111.068,392.961,168.063,47.955,158.931
C09869=1024.883,110.818,392.980,168.061,47.959,158.932
C09870=1024.877,110.569,393.000,168.058,47.963,158.932
C09871=1024.871,110.320,393.020,168.055,47.968,158.933
C09872=1024.866,110.071,393.039,168.052,47.972,158.933
C09873=1024.860,109.821,393.058,168.050,47.976,158.934
C09874=1024.853,109.572,393.077,168.047,47.980,158.934
C09875=1024.848,109.323,393.096,168.045,47.984,158.935
C09876=1024.842,109.073,393.115,168.042,47.988,158.935
C09877=1024.836,108.825,393.134,168.039,47.993,158.935
C09878=1024.831,108.576,393.153,168.037,47.997,158.936
C09879=1024.825,108.327,393.173,168.034,48.001,158.936
C09880=1024.818,108.043,393.194,168.030,48.006,158.937
C09881=1024.811,107.758,393.216,168.027,48.011,158.937
C09882=1024.805,107.473,393.237,168.025,48.016,158.938
C09883=1024.797,107.190,393.259,168.021,48.021,158.938
C09884=1024.792,106.941,393.278,168.018,48.025,158.939
C09885=1024.786,106.691,393.298,168.016,48.029,158.939
C09886=1024.779,106.442,393.316,168.013,48.033,158.940
C09887=1024.774,106.193,393.335,168.011,48.037,158.940
C09888=1024.769,105.944,393.354,168.008,48.041,158.941
C09889=1024.762,105.695,393.373,168.005,48.046,158.941
C09890=1024.757,105.445,393.392,168.003,48.050,158.941
C09891=1024.751,105.196,393.411,168.000,48.054,158.942
C09892=1024.744,104.947,393.430,167.997,48.058,158.942
C09893=1024.739,104.697,393.449,167.995,48.062,158.943
C09894=1024.734,104.449,393.468,167.991,48.067,158.943
C09895=1024.727,104.200,393.487,167.988,48.071,158.944
C09896=1024.722,103.950,393.506,167.986,48.075,158.944
C09897=1024.716,103.700,393.525,167.983,48.079,158.945
C09898=1024.710,103.451,393.543,167.980,48.083,158.945
C09899=1024.705,103.202,393.562,167.978,48.088,158.945
C09900=1024.699,102.953,393.581,167.975,48.092,158.946
C09901=1024.693,102.704,393.600,167.973,48.096,158.946
C09902=1024.687,102.454,393.619,167.970,48.100,158.947
C09903=1024.682,102.206,393.638,167.967,48.105,158.947
C09904=1024.675,101.956,393.657,167.964,48.108,158.948
C09905=1024.670,101.707,393.676,167.962,48.113,158.948
C09906=1024.663,101.458,393.695,167.959,48.117,158.949
C09907=1024.658,101.209,393.714,167.957,48.121,158.949
C09908=1024.653,100.959,393.732,167.954,48.125,158.949
C09909=1024.646,100.710,393.751,167.951,48.129,158.950
C09910=1024.641,100.461,393.770,167.949,48.134,158.950
C09911=1024.636,100.212,393.789,167.946,48.137,158.951
C09912=1024.629,99.963,393.808,167.943,48.142,158.951
C09913=1024.623,99.713,393.827,167.940,48.146,158.952
C09914=1024.618,99.463,393.845,167.938,48.150,158.952
C09915=1024.612,99.215,393.864,167.935,48.154,158.952
C09916=1024.606,98.966,393.882,167.933,48.159,158.953
C09917=1024.600,98.716,393.901,167.930,48.163,158.954
C09918=1024.594,98.466,393.919,167.927,48.167,158.954
C09919=1024.588,98.218,393.938,167.925,48.172,158.954
C09920=1024.582,97.969,393.957,167.922,48.175,158.955
C09921=1024.576,97.719,393.975,167.920,48.180,158.955
C09922=1024.570,97.470,393.994,167.917,48.184,158.956
C09923=1024.565,97.221,394.012,167.914,48.188,158.956
C09924=1024.559,96.971,394.030,167.912,48.193,158.957
C09925=1024.553,96.722,394.050,167.909,48.197,158.957
C09926=1024.547,96.473,394.068,167.907,48.201,158.958
C09927=1024.541,96.224,394.086,167.904,48.205,158.958
C09928=1024.535,95.974,394.105,167.901,48.210,158.959
C09929=1024.529,95.725,394.124,167.899,48.214,158.959
C09930=1024.523,95.476,394.141,167.896,48.218,158.959
C09931=1024.518,95.227,394.161,167.894,48.223,158.960
C09932=1024.512,94.977,394.178,167.891,48.226,158.960
C09933=1024.506,94.729,394.197,167.888,48.231,158.961
C09934=1024.500,94.479,394.216,167.886,48.235,158.961
C09935=1024.494,94.229,394.234,167.883,48.239,158.962
C09936=1024.488,93.981,394.252,167.880,48.243,158.962
C09937=1024.483,93.731,394.271,167.878,48.248,158.963
C09938=1024.476,93.482,394.289,167.875,48.252,158.963
C09939=1024.471,93.233,394.308,167.872,48.256,158.964
C09940=1024.465,92.983,394.326,167.870,48.260,158.964
C09941=1024.459,92.734,394.345,167.867,48.265,158.964
C09942=1024.453,92.485,394.362,167.864,48.268,158.965
C09943=1024.448,92.236,394.382,167.862,48.273,158.965
C09944=1024.441,91.951,394.402,167.858,48.278,158.966
C09945=1024.434,91.667,394.423,167.856,48.282,158.966
C09946=1024.428,91.384,394.444,167.852,48.287,158.967
C09947=1024.421,91.100,394.465,167.850,48.292,158.967
C09948=1024.415,90.850,394.483,167.848,48.296,158.968
C09949=1024.409,90.600,394.502,167.845,48.300,158.968
C09950=1024.404,90.351,394.520,167.842,48.305,158.969
C09951=1024.398,90.102,394.539,167.840,48.309,158.969
C09952=1024.393,89.853,394.557,167.837,48.313,158.970
C09953=1024.386,89.604,394.575,167.834,48.317,158.970
C09954=1024.380,89.354,394.593,167.832,48.322,158.970
C09955=1024.375,89.105,394.611,167.829,48.325,158.971
C09956=1024.368,88.856,394.630,167.827,48.330,158.971
C09957=1024.363,88.607,394.647,167.824,48.335,158.972
C09958=1024.357,88.357,394.665,167.820,48.339,158.972
C09959=1024.351,88.108,394.684,167.818,48.343,158.973
C09960=1024.345,87.859,394.702,167.815,48.348,158.973
C09961=1024.339,87.609,394.720,167.813,48.352,158.974
C09962=1024.333,87.360,394.738,167.810,48.356,158.974
C09963=1024.327,87.111,394.756,167.807,48.360,158.974
C09964=1024.321,86.861,394.774,167.805,48.365,158.975
C09965=1024.316,86.612,394.792,167.802,48.369,158.975
C09966=1024.309,86.363,394.810,167.800,48.373,158.976
C09967=1024.304,86.114,394.828,167.797,48.378,158.976
C09968=1024.298,85.864,394.846,167.794,48.382,158.977
C09969=1024.292,85.616,394.864,167.792,48.386,158.977
C09970=1024.286,85.366,394.882,167.789,48.391,158.978
C09971=1024.280,85.116,394.900,167.787,48.395,158.978
C09972=1024.274,84.867,394.917,167.784,48.399,158.979
C09973=1024.268,84.617,394.935,167.781,48.403,158.979
C09974=1024.262,84.369,394.954,167.779,48.408,158.980
C09975=1024.256,84.119,394.972,167.776,48.411,158.980
C09976=1024.250,83.870,394.989,167.774,48.416,158.980
C09977=1024.244,83.620,395.007,167.771,48.421,158.981
C09978=1024.239,83.372,395.025,167.768,48.424,158.981
C09979=1024.232,83.122,395.043,167.766,48.429,158.982
C09980=1024.227,82.873,395.061,167.763,48.433,158.982
C09981=1024.221,82.623,395.079,167.761,48.437,158.983
C09982=1024.215,82.374,395.096,167.758,48.441,158.983
C09983=1024.209,82.125,395.114,167.755,48.446,158.984
C09984=1024.203,81.876,395.133,167.753,48.450,158.984
C09985=1024.197,81.627,395.150,167.750,48.454,158.984
C09986=1024.192,81.377,395.168,167.747,48.458,158.985
C09987=1024.186,81.128,395.186,167.745,48.463,158.985
C09988=1024.180,80.879,395.204,167.742,48.467,158.986
C09989=1024.174,80.629,395.221,167.740,48.471,158.986
C09990=1024.168,80.380,395.239,167.737,48.476,158.987
C09991=1024.162,80.131,395.258,167.735,48.480,158.987
C09992=1024.156,79.882,395.275,167.732,48.484,158.988
C09993=1024.150,79.632,395.293,167.729,48.488,158.988
C09994=1024.145,79.383,395.311,167.727,48.493,158.989
C09995=1024.139,79.134,395.328,167.724,48.497,158.989
C09996=1024.133,78.884,395.346,167.721,48.501,158.989
//INST
///DATE 2021/06/25 14:49
///ATTR SC,RW,RJ
////FRAME ROBOT
///GROUP1 RB1
NOP
MOVL C00000 V=800.0 PL=0
MOVL C00001 V=800.0 PL=0
MOVL C00002 V=800.0 PL=0
MOVL C00003 V=800.0 PL=0
MOVL C00004 V=800.0 PL=0
MOVL C00005 V=800.0 PL=0
MOVL C00006 V=800.0 PL=0
MOVL C00007 V=800.0 PL=0
MOVL C00008 V=800.0 PL=0
MOVL C00009 V=800.0 PL=0
MOVL C00010 V=800.0 PL=0
MOVL C00011 V=800.0 PL=0
MOVL C00012 V=800.0 PL=0
MOVL C00013 V=800.0 PL=0
MOVL C00014 V=800.0 PL=0
MOVL C00015 V=800.0 PL=0
MOVL C00016 V=800.0 PL=0
MOVL C00017 V=800.0 PL=0
MOVL C00018 V=800.0 PL=0
MOVL C00019 V=800.0 PL=0
MOVL C00020 V=800.0 PL=0
MOVL C00021 V=800.0 PL=0
MOVL C00022 V=800.0 PL=0
MOVL C00023 V=800.0 PL=0
MOVL C00024 V=800.0 PL=0
MOVL C00025 V=800.0 PL=0
MOVL C00026 V=800.0 PL=0
MOVL C00027 V=800.0 PL=0
MOVL C00028 V=800.0 PL=0
MOVL C00029 V=800.0 PL=0
MOVL C00030 V=800.0 PL=0
MOVL C00031 V=800.0 PL=0
MOVL C00032 V=800.0 PL=0
MOVL C00033 V=800.0 PL=0
MOVL C00034 V=800.0 PL=0
MOVL C00035 V=800.0 PL=0
MOVL C00036 V=800.0 PL=0
MOVL C00037 V=800.0 PL=0
MOVL C00038 V=800.0 PL=0
MOVL C00039 V=800.0 PL=0
MOVL C00040 V=800.0 PL=0
MOVL C00041 V=800.0 PL=0
MOVL C00042 V=800.0 PL=0
MOVL C00043 V=800.0 PL=0
MOVL C00044 V=800.0 PL=0
MOVL C00045 V=800.0 PL=0
MOVL C00046 V=800.0 PL=0
MOVL C00047 V=800.0 PL=0
MOVL C00048 V=800.0 PL=0
MOVL C00049 V=800.0 PL=0
MOVL C00050 V=800.0 PL=0
MOVL C00051 V=800.0 PL=0
MOVL C00052 V=800.0 PL=0
MOVL C00053 V=800.0 PL=0
MOVL C00054 V=800.0 PL=0
MOVL C00055 V=800.0 PL=0
MOVL C00056 V=800.0 PL=0
MOVL C00057 V=800.0 PL=0
MOVL C00058 V=800.0 PL=0
MOVL C00059 V=800.0 PL=0
MOVL C00060 V=800.0 PL=0
MOVL C00061 V=800.0 PL=0
MOVL C00062 V=800.0 PL=0
MOVL C00063 V=800.0 PL=0
MOVL C00064 V=800.0 PL=0
MOVL C00065 V=800.0 PL=0
MOVL C00066 V=800.0 PL=0
MOVL C00067 V=800.0 PL=0
MOVL C00068 V=800.0 PL=0
MOVL C00069 V=800.0 PL=0
MOVL C00070 V=800.0 PL=0
MOVL C00071 V=800.0 PL=0
MOVL C00072 V=800.0 PL=0
MOVL C00073 V=800.0 PL=0
MOVL C00074 V=800.0 PL=0
MOVL C00075 V=800.0 PL=0
MOVL C00076 V=800.0 PL=0
MOVL C00077 V=800.0 PL=0
MOVL C00078 V=800.0 PL=0
MOVL C00079 V=800.0 PL=0
MOVL C00080 V=800.0 PL=0
MOVL C00081 V=800.0 PL=0
MOVL C00082 V=800.0 PL=0
MOVL C00083 V=800.0 PL=0
MOVL C00084 V=800.0 PL=0
MOVL C00085 V=800.0 PL=0
MOVL C00086 V=800.0 PL=0
MOVL C00087 V=800.0 PL=0
MOVL C00088 V=800.0 PL=0
MOVL C00089 V=800.0 PL=0
MOVL C00090 V=800.0 PL=0
MOVL C00091 V=800.0 PL=0
MOVL C00092 V=800.0 PL=0
MOVL C00093 V=800.0 PL=0
MOVL C00094 V=800.0 PL=0
MOVL C00095 V=800.0 PL=0
MOVL C00096 V=800.0 PL=0
MOVL C00097 V=800.0 PL=0
MOVL C00098 V=800.0 PL=0
MOVL C00099 V=800.0 PL=0
MOVL C00100 V=800.0 PL=0
MOVL C00101 V=800.0 PL=0
MOVL C00102 V=800.0 PL=0
MOVL C00103 V=800.0 PL=0
MOVL C00104 V=800.0 PL=0
MOVL C00105 V=800.0 PL=0
MOVL C00106 V=800.0 PL=0
MOVL C00107 V=800.0 PL=0
MOVL C00108 V=800.0 PL=0
MOVL C00109 V=800.0 PL=0
MOVL C00110 V=800.0 PL=0
MOVL C00111 V=800.0 PL=0
MOVL C00112 V=800.0 PL=0
MOVL C00113 V=800.0 PL=0
MOVL C00114 V=800.0 PL=0
MOVL C00115 V=800.0 PL=0
MOVL C00116 V=800.0 PL=0
MOVL C00117 V=800.0 PL=0
MOVL C00118 V=800.0 PL=0
MOVL C00119 V=800.0 PL=0
MOVL C00120 V=800.0 PL=0
MOVL C00121 V=800.0 PL=0
MOVL C00122 V=800.0 PL=0
MOVL C00123 V=800.0 PL=0
MOVL C00124 V=800.0 PL=0
MOVL C00125 V=800.0 PL=0
MOVL C00126 V=800.0 PL=0
MOVL C00127 V=800.0 PL=0
MOVL C00128 V=800.0 PL=0
MOVL C00129 V=800.0 PL=0
MOVL C00130 V=800.0 PL=0
MOVL C00131 V=800.0 PL=0
MOVL C00132 V=800.0 PL=0
MOVL C00133 V=800.0 PL=0
MOVL C00134 V=800.0 PL=0
MOVL C00135 V=800.0 PL=0
MOVL C00136 V=800.0 PL=0
MOVL C00137 V=800.0 PL=0
MOVL C00138 V=800.0 PL=0
MOVL C00139 V=800.0 PL=0
MOVL C00140 V=800.0 PL=0
MOVL C00141 V=800.0 PL=0
MOVL C00142 V=800.0 PL=0
MOVL C00143 V=800.0 PL=0
MOVL C00144 V=800.0 PL=0
MOVL C00145 V=800.0 PL=0
MOVL C00146 V=800.0 PL=0
MOVL C00147 V=800.0 PL=0
MOVL C00148 V=800.0 PL=0
MOVL C00149 V=800.0 PL=0
MOVL C00150 V=800.0 PL=0
MOVL C00151 V=800.0 PL=0
MOVL C00152 V=800.0 PL=0
MOVL C00153 V=800.0 PL=0
MOVL C00154 V=800.0 PL=0
MOVL C00155 V=800.0 PL=0
MOVL C00156 V=800.0 PL=0
MOVL C00157 V=800.0 PL=0
MOVL C00158 V=800.0 PL=0
MOVL C00159 V=800.0 PL=0
MOVL C00160 V=800.0 PL=0
MOVL C00161 V=800.0 PL=0
MOVL C00162 V=800.0 PL=0
MOVL C00163 V=800.0 PL=0
MOVL C00164 V=800.0 PL=0
MOVL C00165 V=800.0 PL=0
MOVL C00166 V=800.0 PL=0
MOVL C00167 V=800.0 PL=0
MOVL C00168 V=800.0 PL=0
MOVL C00169 V=800.0 PL=0
MOVL C00170 V=800.0 PL=0
MOVL C00171 V=800.0 PL=0
MOVL C00172 V=800.0 PL=0
MOVL C00173 V=800.0 PL=0
MOVL C00174 V=800.0 PL=0
MOVL C00175 V=800.0 PL=0
MOVL C00176 V=800.0 PL=0
MOVL C00177 V=800.0 PL=0
MOVL C00178 V=800.0 PL=0
MOVL C00179 V=800.0 PL=0
MOVL C00180 V=800.0 PL=0
MOVL C00181 V=800.0 PL=0
MOVL C00182 V=800.0 PL=0
MOVL C00183 V=800.0 PL=0
MOVL C00184 V=800.0 PL=0
MOVL C00185 V=800.0 PL=0
MOVL C00186 V=800.0 PL=0
MOVL C00187 V=800.0 PL=0
MOVL C00188 V=800.0 PL=0
MOVL C00189 V=800.0 PL=0
MOVL C00190 V=800.0 PL=0
MOVL C00191 V=800.0 PL=0
MOVL C00192 V=800.0 PL=0
MOVL C00193 V=800.0 PL=0
MOVL C00194 V=800.0 PL=0
MOVL C00195 V=800.0 PL=0
MOVL C00196 V=800.0 PL=0
MOVL C00197 V=800.0 PL=0
MOVL C00198 V=800.0 PL=0
MOVL C00199 V=800.0 PL=0
MOVL C00200 V=800.0 PL=0
MOVL C00201 V=800.0 PL=0
MOVL C00202 V=800.0 PL=0
MOVL C00203 V=800.0 PL=0
MOVL C00204 V=800.0 PL=0
MOVL C00205 V=800.0 PL=0
MOVL C00206 V=800.0 PL=0
MOVL C00207 V=800.0 PL=0
MOVL C00208 V=800.0 PL=0
MOVL C00209 V=800.0 PL=0
MOVL C00210 V=800.0 PL=0
MOVL C00211 V=800.0 PL=0
MOVL C00212 V=800.0 PL=0
MOVL C00213 V=800.0 PL=0
MOVL C00214 V=800.0 PL=0
MOVL C00215 V=800.0 PL=0
MOVL C00216 V=800.0 PL=0
MOVL C00217 V=800.0 PL=0
MOVL C00218 V=800.0 PL=0
MOVL C00219 V=800.0 PL=0
MOVL C00220 V=800.0 PL=0
MOVL C00221 V=800.0 PL=0
MOVL C00222 V=800.0 PL=0
MOVL C00223 V=800.0 PL=0
MOVL C00224 V=800.0 PL=0
MOVL C00225 V=800.0 PL=0
MOVL C00226 V=800.0 PL=0
MOVL C00227 V=800.0 PL=0
MOVL C00228 V=800.0 PL=0
MOVL C00229 V=800.0 PL=0
MOVL C00230 V=800.0 PL=0
MOVL C00231 V=800.0 PL=0
MOVL C00232 V=800.0 PL=0
MOVL C00233 V=800.0 PL=0
MOVL C00234 V=800.0 PL=0
MOVL C00235 V=800.0 PL=0
MOVL C00236 V=800.0 PL=0
MOVL C00237 V=800.0 PL=0
MOVL C00238 V=800.0 PL=0
MOVL C00239 V=800.0 PL=0
MOVL C00240 V=800.0 PL=0
MOVL C00241 V=800.0 PL=0
MOVL C00242 V=800.0 PL=0
MOVL C00243 V=800.0 PL=0
MOVL C00244 V=800.0 PL=0
MOVL C00245 V=800.0 PL=0
MOVL C00246 V=800.0 PL=0
MOVL C00247 V=800.0 PL=0
MOVL C00248 V=800.0 PL=0
MOVL C00249 V=800.0 PL=0
MOVL C00250 V=800.0 PL=0
MOVL C00251 V=800.0 PL=0
MOVL C00252 V=800.0 PL=0
MOVL C00253 V=800.0 PL=0
MOVL C00254 V=800.0 PL=0
MOVL C00255 V=800.0 PL=0
MOVL C00256 V=800.0 PL=0
MOVL C00257 V=800.0 PL=0
MOVL C00258 V=800.0 PL=0
MOVL C00259 V=800.0 PL=0
MOVL C00260 V=800.0 PL=0
MOVL C00261 V=800.0 PL=0
MOVL C00262 V=800.0 PL=0
MOVL C00263 V=800.0 PL=0
MOVL C00264 V=800.0 PL=0
MOVL C00265 V=800.0 PL=0
MOVL C00266 V=800.0 PL=0
MOVL C00267 V=800.0 PL=0
MOVL C00268 V=800.0 PL=0
MOVL C00269 V=800.0 PL=0
MOVL C00270 V=800.0 PL=0
MOVL C00271 V=800.0 PL=0
MOVL C00272 V=800.0 PL=0
MOVL C00273 V=800.0 PL=0
MOVL C00274 V=800.0 PL=0
MOVL C00275 V=800.0 PL=0
MOVL C00276 V=800.0 PL=0
MOVL C00277 V=800.0 PL=0
MOVL C00278 V=800.0 PL=0
MOVL C00279 V=800.0 PL=0
MOVL C00280 V=800.0 PL=0
MOVL C00281 V=800.0 PL=0
MOVL C00282 V=800.0 PL=0
MOVL C00283 V=800.0 PL=0
MOVL C00284 V=800.0 PL=0
MOVL C00285 V=800.0 PL=0
MOVL C00286 V=800.0 PL=0
MOVL C00287 V=800.0 PL=0
MOVL C00288 V=800.0 PL=0
MOVL C00289 V=800.0 PL=0
MOVL C00290 V=800.0 PL=0
MOVL C00291 V=800.0 PL=0
MOVL C00292 V=800.0 PL=0
MOVL C00293 V=800.0 PL=0
MOVL C00294 V=800.0 PL=0
MOVL C00295 V=800.0 PL=0
MOVL C00296 V=800.0 PL=0
MOVL C00297 V=800.0 PL=0
MOVL C00298 V=800.0 PL=0
MOVL C00299 V=800.0 PL=0
MOVL C00300 V=800.0 PL=0
MOVL C00301 V=800.0 PL=0
MOVL C00302 V=800.0 PL=0
MOVL C00303 V=800.0 PL=0
MOVL C00304 V=800.0 PL=0
MOVL C00305 V=800.0 PL=0
MOVL C00306 V=800.0 PL=0
MOVL C00307 V=800.0 PL=0
MOVL C00308 V=800.0 PL=0
MOVL C00309 V=800.0 PL=0
MOVL C00310 V=800.0 PL=0
MOVL C00311 V=800.0 PL=0
MOVL C00312 V=800.0 PL=0
MOVL C00313 V=800.0 PL=0
MOVL C00314 V=800.0 PL=0
MOVL C00315 V=800.0 PL=0
MOVL C00316 V=800.0 PL=0
MOVL C00317 V=800.0 PL=0
MOVL C00318 V=800.0 PL=0
MOVL C00319 V=800.0 PL=0
MOVL C00320 V=800.0 PL=0
MOVL C00321 V=800.0 PL=0
MOVL C00322 V=800.0 PL=0
MOVL C00323 V=800.0 PL=0
MOVL C00324 V=800.0 PL=0
MOVL C00325 V=800.0 PL=0
MOVL C00326 V=800.0 PL=0
MOVL C00327 V=800.0 PL=0
MOVL C00328 V=800.0 PL=0
MOVL C00329 V=800.0 PL=0
MOVL C00330 V=800.0 PL=0
MOVL C00331 V=800.0 PL=0
MOVL C00332 V=800.0 PL=0
MOVL C00333 V=800.0 PL=0
MOVL C00334 V=800.0 PL=0
MOVL C00335 V=800.0 PL=0
MOVL C00336 V=800.0 PL=0
MOVL C00337 V=800.0 PL=0
MOVL C00338 V=800.0 PL=0
MOVL C00339 V=800.0 PL=0
MOVL C00340 V=800.0 PL=0
MOVL C00341 V=800.0 PL=0
MOVL C00342 V=800.0 PL=0
MOVL C00343 V=800.0 PL=0
MOVL C00344 V=800.0 PL=0
MOVL C00345 V=800.0 PL=0
MOVL C00346 V=800.0 PL=0
MOVL C00347 V=800.0 PL=0
MOVL C00348 V=800.0 PL=0
MOVL C00349 V=800.0 PL=0
MOVL C00350 V=800.0 PL=0
MOVL C00351 V=800.0 PL=0
MOVL C00352 V=800.0 PL=0
MOVL C00353 V=800.0 PL=0
MOVL C00354 V=800.0 PL=0
MOVL C00355 V=800.0 PL=0
MOVL C00356 V=800.0 PL=0
MOVL C00357 V=800.0 PL=0
MOVL C00358 V=800.0 PL=0
MOVL C00359 V=800.0 PL=0
MOVL C00360 V=800.0 PL=0
MOVL C00361 V=800.0 PL=0
MOVL C00362 V=800.0 PL=0
MOVL C00363 V=800.0 PL=0
MOVL C00364 V=800.0 PL=0
MOVL C00365 V=800.0 PL=0
MOVL C00366 V=800.0 PL=0
MOVL C00367 V=800.0 PL=0
MOVL C00368 V=800.0 PL=0
MOVL C00369 V=800.0 PL=0
MOVL C00370 V=800.0 PL=0
MOVL C00371 V=800.0 PL=0
MOVL C00372 V=800.0 PL=0
MOVL C00373 V=800.0 PL=0
MOVL C00374 V=800.0 PL=0
MOVL C00375 V=800.0 PL=0
MOVL C00376 V=800.0 PL=0
MOVL C00377 V=800.0 PL=0
MOVL C00378 V=800.0 PL=0
MOVL C00379 V=800.0 PL=0
MOVL C00380 V=800.0 PL=0
MOVL C00381 V=800.0 PL=0
MOVL C00382 V=800.0 PL=0
MOVL C00383 V=800.0 PL=0
MOVL C00384 V=800.0 PL=0
MOVL C00385 V=800.0 PL=0
MOVL C00386 V=800.0 PL=0
MOVL C00387 V=800.0 PL=0
MOVL C00388 V=800.0 PL=0
MOVL C00389 V=800.0 PL=0
MOVL C00390 V=800.0 PL=0
MOVL C00391 V=800.0 PL=0
MOVL C00392 V=800.0 PL=0
MOVL C00393 V=800.0 PL=0
MOVL C00394 V=800.0 PL=0
MOVL C00395 V=800.0 PL=0
MOVL C00396 V=800.0 PL=0
MOVL C00397 V=800.0 PL=0
MOVL C00398 V=800.0 PL=0
MOVL C00399 V=800.0 PL=0
MOVL C00400 V=800.0 PL=0
MOVL C00401 V=800.0 PL=0
MOVL C00402 V=800.0 PL=0
MOVL C00403 V=800.0 PL=0
MOVL C00404 V=800.0 PL=0
MOVL C00405 V=800.0 PL=0
MOVL C00406 V=800.0 PL=0
MOVL C00407 V=800.0 PL=0
MOVL C00408 V=800.0 PL=0
MOVL C00409 V=800.0 PL=0
MOVL C00410 V=800.0 PL=0
MOVL C00411 V=800.0 PL=0
MOVL C00412 V=800.0 PL=0
MOVL C00413 V=800.0 PL=0
MOVL C00414 V=800.0 PL=0
MOVL C00415 V=800.0 PL=0
MOVL C00416 V=800.0 PL=0
MOVL C00417 V=800.0 PL=0
MOVL C00418 V=800.0 PL=0
MOVL C00419 V=800.0 PL=0
MOVL C00420 V=800.0 PL=0
MOVL C00421 V=800.0 PL=0
MOVL C00422 V=800.0 PL=0
MOVL C00423 V=800.0 PL=0
MOVL C00424 V=800.0 PL=0
MOVL C00425 V=800.0 PL=0
MOVL C00426 V=800.0 PL=0
MOVL C00427 V=800.0 PL=0
MOVL C00428 V=800.0 PL=0
MOVL C00429 V=800.0 PL=0
MOVL C00430 V=800.0 PL=0
MOVL C00431 V=800.0 PL=0
MOVL C00432 V=800.0 PL=0
MOVL C00433 V=800.0 PL=0
MOVL C00434 V=800.0 PL=0
MOVL C00435 V=800.0 PL=0
MOVL C00436 V=800.0 PL=0
MOVL C00437 V=800.0 PL=0
MOVL C00438 V=800.0 PL=0
MOVL C00439 V=800.0 PL=0
MOVL C00440 V=800.0 PL=0
MOVL C00441 V=800.0 PL=0
MOVL C00442 V=800.0 PL=0
MOVL C00443 V=800.0 PL=0
MOVL C00444 V=800.0 PL=0
MOVL C00445 V=800.0 PL=0
MOVL C00446 V=800.0 PL=0
MOVL C00447 V=800.0 PL=0
MOVL C00448 V=800.0 PL=0
MOVL C00449 V=800.0 PL=0
MOVL C00450 V=800.0 PL=0
MOVL C00451 V=800.0 PL=0
MOVL C00452 V=800.0 PL=0
MOVL C00453 V=800.0 PL=0
MOVL C00454 V=800.0 PL=0
MOVL C00455 V=800.0 PL=0
MOVL C00456 V=800.0 PL=0
MOVL C00457 V=800.0 PL=0
MOVL C00458 V=800.0 PL=0
MOVL C00459 V=800.0 PL=0
MOVL C00460 V=800.0 PL=0
MOVL C00461 V=800.0 PL=0
MOVL C00462 V=800.0 PL=0
MOVL C00463 V=800.0 PL=0
MOVL C00464 V=800.0 PL=0
MOVL C00465 V=800.0 PL=0
MOVL C00466 V=800.0 PL=0
MOVL C00467 V=800.0 PL=0
MOVL C00468 V=800.0 PL=0
MOVL C00469 V=800.0 PL=0
MOVL C00470 V=800.0 PL=0
MOVL C00471 V=800.0 PL=0
MOVL C00472 V=800.0 PL=0
MOVL C00473 V=800.0 PL=0
MOVL C00474 V=800.0 PL=0
MOVL C00475 V=800.0 PL=0
MOVL C00476 V=800.0 PL=0
MOVL C00477 V=800.0 PL=0
MOVL C00478 V=800.0 PL=0
MOVL C00479 V=800.0 PL=0
MOVL C00480 V=800.0 PL=0
MOVL C00481 V=800.0 PL=0
MOVL C00482 V=800.0 PL=0
MOVL C00483 V=800.0 PL=0
MOVL C00484 V=800.0 PL=0
MOVL C00485 V=800.0 PL=0
MOVL C00486 V=800.0 PL=0
MOVL C00487 V=800.0 PL=0
MOVL C00488 V=800.0 PL=0
MOVL C00489 V=800.0 PL=0
MOVL C00490 V=800.0 PL=0
MOVL C00491 V=800.0 PL=0
MOVL C00492 V=800.0 PL=0
MOVL C00493 V=800.0 PL=0
MOVL C00494 V=800.0 PL=0
MOVL C00495 V=800.0 PL=0
MOVL C00496 V=800.0 PL=0
MOVL C00497 V=800.0 PL=0
MOVL C00498 V=800.0 PL=0
MOVL C00499 V=800.0 PL=0
MOVL C00500 V=800.0 PL=0
MOVL C00501 V=800.0 PL=0
MOVL C00502 V=800.0 PL=0
MOVL C00503 V=800.0 PL=0
MOVL C00504 V=800.0 PL=0
MOVL C00505 V=800.0 PL=0
MOVL C00506 V=800.0 PL=0
MOVL C00507 V=800.0 PL=0
MOVL C00508 V=800.0 PL=0
MOVL C00509 V=800.0 PL=0
MOVL C00510 V=800.0 PL=0
MOVL C00511 V=800.0 PL=0
MOVL C00512 V=800.0 PL=0
MOVL C00513 V=800.0 PL=0
MOVL C00514 V=800.0 PL=0
MOVL C00515 V=800.0 PL=0
MOVL C00516 V=800.0 PL=0
MOVL C00517 V=800.0 PL=0
MOVL C00518 V=800.0 PL=0
MOVL C00519 V=800.0 PL=0
MOVL C00520 V=800.0 PL=0
MOVL C00521 V=800.0 PL=0
MOVL C00522 V=800.0 PL=0
MOVL C00523 V=800.0 PL=0
MOVL C00524 V=800.0 PL=0
MOVL C00525 V=800.0 PL=0
MOVL C00526 V=800.0 PL=0
MOVL C00527 V=800.0 PL=0
MOVL C00528 V=800.0 PL=0
MOVL C00529 V=800.0 PL=0
MOVL C00530 V=800.0 PL=0
MOVL C00531 V=800.0 PL=0
MOVL C00532 V=800.0 PL=0
MOVL C00533 V=800.0 PL=0
MOVL C00534 V=800.0 PL=0
MOVL C00535 V=800.0 PL=0
MOVL C00536 V=800.0 PL=0
MOVL C00537 V=800.0 PL=0
MOVL C00538 V=800.0 PL=0
MOVL C00539 V=800.0 PL=0
MOVL C00540 V=800.0 PL=0
MOVL C00541 V=800.0 PL=0
MOVL C00542 V=800.0 PL=0
MOVL C00543 V=800.0 PL=0
MOVL C00544 V=800.0 PL=0
MOVL C00545 V=800.0 PL=0
MOVL C00546 V=800.0 PL=0
MOVL C00547 V=800.0 PL=0
MOVL C00548 V=800.0 PL=0
MOVL C00549 V=800.0 PL=0
MOVL C00550 V=800.0 PL=0
MOVL C00551 V=800.0 PL=0
MOVL C00552 V=800.0 PL=0
MOVL C00553 V=800.0 PL=0
MOVL C00554 V=800.0 PL=0
MOVL C00555 V=800.0 PL=0
MOVL C00556 V=800.0 PL=0
MOVL C00557 V=800.0 PL=0
MOVL C00558 V=800.0 PL=0
MOVL C00559 V=800.0 PL=0
MOVL C00560 V=800.0 PL=0
MOVL C00561 V=800.0 PL=0
MOVL C00562 V=800.0 PL=0
MOVL C00563 V=800.0 PL=0
MOVL C00564 V=800.0 PL=0
MOVL C00565 V=800.0 PL=0
MOVL C00566 V=800.0 PL=0
MOVL C00567 V=800.0 PL=0
MOVL C00568 V=800.0 PL=0
MOVL C00569 V=800.0 PL=0
MOVL C00570 V=800.0 PL=0
MOVL C00571 V=800.0 PL=0
MOVL C00572 V=800.0 PL=0
MOVL C00573 V=800.0 PL=0
MOVL C00574 V=800.0 PL=0
MOVL C00575 V=800.0 PL=0
MOVL C00576 V=800.0 PL=0
MOVL C00577 V=800.0 PL=0
MOVL C00578 V=800.0 PL=0
MOVL C00579 V=800.0 PL=0
MOVL C00580 V=800.0 PL=0
MOVL C00581 V=800.0 PL=0
MOVL C00582 V=800.0 PL=0
MOVL C00583 V=800.0 PL=0
MOVL C00584 V=800.0 PL=0
MOVL C00585 V=800.0 PL=0
MOVL C00586 V=800.0 PL=0
MOVL C00587 V=800.0 PL=0
MOVL C00588 V=800.0 PL=0
MOVL C00589 V=800.0 PL=0
MOVL C00590 V=800.0 PL=0
MOVL C00591 V=800.0 PL=0
MOVL C00592 V=800.0 PL=0
MOVL C00593 V=800.0 PL=0
MOVL C00594 V=800.0 PL=0
MOVL C00595 V=800.0 PL=0
MOVL C00596 V=800.0 PL=0
MOVL C00597 V=800.0 PL=0
MOVL C00598 V=800.0 PL=0
MOVL C00599 V=800.0 PL=0
MOVL C00600 V=800.0 PL=0
MOVL C00601 V=800.0 PL=0
MOVL C00602 V=800.0 PL=0
MOVL C00603 V=800.0 PL=0
MOVL C00604 V=800.0 PL=0
MOVL C00605 V=800.0 PL=0
MOVL C00606 V=800.0 PL=0
MOVL C00607 V=800.0 PL=0
MOVL C00608 V=800.0 PL=0
MOVL C00609 V=800.0 PL=0
MOVL C00610 V=800.0 PL=0
MOVL C00611 V=800.0 PL=0
MOVL C00612 V=800.0 PL=0
MOVL C00613 V=800.0 PL=0
MOVL C00614 V=800.0 PL=0
MOVL C00615 V=800.0 PL=0
MOVL C00616 V=800.0 PL=0
MOVL C00617 V=800.0 PL=0
MOVL C00618 V=800.0 PL=0
MOVL C00619 V=800.0 PL=0
MOVL C00620 V=800.0 PL=0
MOVL C00621 V=800.0 PL=0
MOVL C00622 V=800.0 PL=0
MOVL C00623 V=800.0 PL=0
MOVL C00624 V=800.0 PL=0
MOVL C00625 V=800.0 PL=0
MOVL C00626 V=800.0 PL=0
MOVL C00627 V=800.0 PL=0
MOVL C00628 V=800.0 PL=0
MOVL C00629 V=800.0 PL=0
MOVL C00630 V=800.0 PL=0
MOVL C00631 V=800.0 PL=0
MOVL C00632 V=800.0 PL=0
MOVL C00633 V=800.0 PL=0
MOVL C00634 V=800.0 PL=0
MOVL C00635 V=800.0 PL=0
MOVL C00636 V=800.0 PL=0
MOVL C00637 V=800.0 PL=0
MOVL C00638 V=800.0 PL=0
MOVL C00639 V=800.0 PL=0
MOVL C00640 V=800.0 PL=0
MOVL C00641 V=800.0 PL=0
MOVL C00642 V=800.0 PL=0
MOVL C00643 V=800.0 PL=0
MOVL C00644 V=800.0 PL=0
MOVL C00645 V=800.0 PL=0
MOVL C00646 V=800.0 PL=0
MOVL C00647 V=800.0 PL=0
MOVL C00648 V=800.0 PL=0
MOVL C00649 V=800.0 PL=0
MOVL C00650 V=800.0 PL=0
MOVL C00651 V=800.0 PL=0
MOVL C00652 V=800.0 PL=0
MOVL C00653 V=800.0 PL=0
MOVL C00654 V=800.0 PL=0
MOVL C00655 V=800.0 PL=0
MOVL C00656 V=800.0 PL=0
MOVL C00657 V=800.0 PL=0
MOVL C00658 V=800.0 PL=0
MOVL C00659 V=800.0 PL=0
MOVL C00660 V=800.0 PL=0
MOVL C00661 V=800.0 PL=0
MOVL C00662 V=800.0 PL=0
MOVL C00663 V=800.0 PL=0
MOVL C00664 V=800.0 PL=0
MOVL C00665 V=800.0 PL=0
MOVL C00666 V=800.0 PL=0
MOVL C00667 V=800.0 PL=0
MOVL C00668 V=800.0 PL=0
MOVL C00669 V=800.0 PL=0
MOVL C00670 V=800.0 PL=0
MOVL C00671 V=800.0 PL=0
MOVL C00672 V=800.0 PL=0
MOVL C00673 V=800.0 PL=0
MOVL C00674 V=800.0 PL=0
MOVL C00675 V=800.0 PL=0
MOVL C00676 V=800.0 PL=0
MOVL C00677 V=800.0 PL=0
MOVL C00678 V=800.0 PL=0
MOVL C00679 V=800.0 PL=0
MOVL C00680 V=800.0 PL=0
MOVL C00681 V=800.0 PL=0
MOVL C00682 V=800.0 PL=0
MOVL C00683 V=800.0 PL=0
MOVL C00684 V=800.0 PL=0
MOVL C00685 V=800.0 PL=0
MOVL C00686 V=800.0 PL=0
MOVL C00687 V=800.0 PL=0
MOVL C00688 V=800.0 PL=0
MOVL C00689 V=800.0 PL=0
MOVL C00690 V=800.0 PL=0
MOVL C00691 V=800.0 PL=0
MOVL C00692 V=800.0 PL=0
MOVL C00693 V=800.0 PL=0
MOVL C00694 V=800.0 PL=0
MOVL C00695 V=800.0 PL=0
MOVL C00696 V=800.0 PL=0
MOVL C00697 V=800.0 PL=0
MOVL C00698 V=800.0 PL=0
MOVL C00699 V=800.0 PL=0
MOVL C00700 V=800.0 PL=0
MOVL C00701 V=800.0 PL=0
MOVL C00702 V=800.0 PL=0
MOVL C00703 V=800.0 PL=0
MOVL C00704 V=800.0 PL=0
MOVL C00705 V=800.0 PL=0
MOVL C00706 V=800.0 PL=0
MOVL C00707 V=800.0 PL=0
MOVL C00708 V=800.0 PL=0
MOVL C00709 V=800.0 PL=0
MOVL C00710 V=800.0 PL=0
MOVL C00711 V=800.0 PL=0
MOVL C00712 V=800.0 PL=0
MOVL C00713 V=800.0 PL=0
MOVL C00714 V=800.0 PL=0
MOVL C00715 V=800.0 PL=0
MOVL C00716 V=800.0 PL=0
MOVL C00717 V=800.0 PL=0
MOVL C00718 V=800.0 PL=0
MOVL C00719 V=800.0 PL=0
MOVL C00720 V=800.0 PL=0
MOVL C00721 V=800.0 PL=0
MOVL C00722 V=800.0 PL=0
MOVL C00723 V=800.0 PL=0
MOVL C00724 V=800.0 PL=0
MOVL C00725 V=800.0 PL=0
MOVL C00726 V=800.0 PL=0
MOVL C00727 V=800.0 PL=0
MOVL C00728 V=800.0 PL=0
MOVL C00729 V=800.0 PL=0
MOVL C00730 V=800.0 PL=0
MOVL C00731 V=800.0 PL=0
MOVL C00732 V=800.0 PL=0
MOVL C00733 V=800.0 PL=0
MOVL C00734 V=800.0 PL=0
MOVL C00735 V=800.0 PL=0
MOVL C00736 V=800.0 PL=0
MOVL C00737 V=800.0 PL=0
MOVL C00738 V=800.0 PL=0
MOVL C00739 V=800.0 PL=0
MOVL C00740 V=800.0 PL=0
MOVL C00741 V=800.0 PL=0
MOVL C00742 V=800.0 PL=0
MOVL C00743 V=800.0 PL=0
MOVL C00744 V=800.0 PL=0
MOVL C00745 V=800.0 PL=0
MOVL C00746 V=800.0 PL=0
MOVL C00747 V=800.0 PL=0
MOVL C00748 V=800.0 PL=0
MOVL C00749 V=800.0 PL=0
MOVL C00750 V=800.0 PL=0
MOVL C00751 V=800.0 PL=0
MOVL C00752 V=800.0 PL=0
MOVL C00753 V=800.0 PL=0
MOVL C00754 V=800.0 PL=0
MOVL C00755 V=800.0 PL=0
MOVL C00756 V=800.0 PL=0
MOVL C00757 V=800.0 PL=0
MOVL C00758 V=800.0 PL=0
MOVL C00759 V=800.0 PL=0
MOVL C00760 V=800.0 PL=0
MOVL C00761 V=800.0 PL=0
MOVL C00762 V=800.0 PL=0
MOVL C00763 V=800.0 PL=0
MOVL C00764 V=800.0 PL=0
MOVL C00765 V=800.0 PL=0
MOVL C00766 V=800.0 PL=0
MOVL C00767 V=800.0 PL=0
MOVL C00768 V=800.0 PL=0
MOVL C00769 V=800.0 PL=0
MOVL C00770 V=800.0 PL=0
MOVL C00771 V=800.0 PL=0
MOVL C00772 V=800.0 PL=0
MOVL C00773 V=800.0 PL=0
MOVL C00774 V=800.0 PL=0
MOVL C00775 V=800.0 PL=0
MOVL C00776 V=800.0 PL=0
MOVL C00777 V=800.0 PL=0
MOVL C00778 V=800.0 PL=0
MOVL C00779 V=800.0 PL=0
MOVL C00780 V=800.0 PL=0
MOVL C00781 V=800.0 PL=0
MOVL C00782 V=800.0 PL=0
MOVL C00783 V=800.0 PL=0
MOVL C00784 V=800.0 PL=0
MOVL C00785 V=800.0 PL=0
MOVL C00786 V=800.0 PL=0
MOVL C00787 V=800.0 PL=0
MOVL C00788 V=800.0 PL=0
MOVL C00789 V=800.0 PL=0
MOVL C00790 V=800.0 PL=0
MOVL C00791 V=800.0 PL=0
MOVL C00792 V=800.0 PL=0
MOVL C00793 V=800.0 PL=0
MOVL C00794 V=800.0 PL=0
MOVL C00795 V=800.0 PL=0
MOVL C00796 V=800.0 PL=0
MOVL C00797 V=800.0 PL=0
MOVL C00798 V=800.0 PL=0
MOVL C00799 V=800.0 PL=0
MOVL C00800 V=800.0 PL=0
MOVL C00801 V=800.0 PL=0
MOVL C00802 V=800.0 PL=0
MOVL C00803 V=800.0 PL=0
MOVL C00804 V=800.0 PL=0
MOVL C00805 V=800.0 PL=0
MOVL C00806 V=800.0 PL=0
MOVL C00807 V=800.0 PL=0
MOVL C00808 V=800.0 PL=0
MOVL C00809 V=800.0 PL=0
MOVL C00810 V=800.0 PL=0
MOVL C00811 V=800.0 PL=0
MOVL C00812 V=800.0 PL=0
MOVL C00813 V=800.0 PL=0
MOVL C00814 V=800.0 PL=0
MOVL C00815 V=800.0 PL=0
MOVL C00816 V=800.0 PL=0
MOVL C00817 V=800.0 PL=0
MOVL C00818 V=800.0 PL=0
MOVL C00819 V=800.0 PL=0
MOVL C00820 V=800.0 PL=0
MOVL C00821 V=800.0 PL=0
MOVL C00822 V=800.0 PL=0
MOVL C00823 V=800.0 PL=0
MOVL C00824 V=800.0 PL=0
MOVL C00825 V=800.0 PL=0
MOVL C00826 V=800.0 PL=0
MOVL C00827 V=800.0 PL=0
MOVL C00828 V=800.0 PL=0
MOVL C00829 V=800.0 PL=0
MOVL C00830 V=800.0 PL=0
MOVL C00831 V=800.0 PL=0
MOVL C00832 V=800.0 PL=0
MOVL C00833 V=800.0 PL=0
MOVL C00834 V=800.0 PL=0
MOVL C00835 V=800.0 PL=0
MOVL C00836 V=800.0 PL=0
MOVL C00837 V=800.0 PL=0
MOVL C00838 V=800.0 PL=0
MOVL C00839 V=800.0 PL=0
MOVL C00840 V=800.0 PL=0
MOVL C00841 V=800.0 PL=0
MOVL C00842 V=800.0 PL=0
MOVL C00843 V=800.0 PL=0
MOVL C00844 V=800.0 PL=0
MOVL C00845 V=800.0 PL=0
MOVL C00846 V=800.0 PL=0
MOVL C00847 V=800.0 PL=0
MOVL C00848 V=800.0 PL=0
MOVL C00849 V=800.0 PL=0
MOVL C00850 V=800.0 PL=0
MOVL C00851 V=800.0 PL=0
MOVL C00852 V=800.0 PL=0
MOVL C00853 V=800.0 PL=0
MOVL C00854 V=800.0 PL=0
MOVL C00855 V=800.0 PL=0
MOVL C00856 V=800.0 PL=0
MOVL C00857 V=800.0 PL=0
MOVL C00858 V=800.0 PL=0
MOVL C00859 V=800.0 PL=0
MOVL C00860 V=800.0 PL=0
MOVL C00861 V=800.0 PL=0
MOVL C00862 V=800.0 PL=0
MOVL C00863 V=800.0 PL=0
MOVL C00864 V=800.0 PL=0
MOVL C00865 V=800.0 PL=0
MOVL C00866 V=800.0 PL=0
MOVL C00867 V=800.0 PL=0
MOVL C00868 V=800.0 PL=0
MOVL C00869 V=800.0 PL=0
MOVL C00870 V=800.0 PL=0
MOVL C00871 V=800.0 PL=0
MOVL C00872 V=800.0 PL=0
MOVL C00873 V=800.0 PL=0
MOVL C00874 V=800.0 PL=0
MOVL C00875 V=800.0 PL=0
MOVL C00876 V=800.0 PL=0
MOVL C00877 V=800.0 PL=0
MOVL C00878 V=800.0 PL=0
MOVL C00879 V=800.0 PL=0
MOVL C00880 V=800.0 PL=0
MOVL C00881 V=800.0 PL=0
MOVL C00882 V=800.0 PL=0
MOVL C00883 V=800.0 PL=0
MOVL C00884 V=800.0 PL=0
MOVL C00885 V=800.0 PL=0
MOVL C00886 V=800.0 PL=0
MOVL C00887 V=800.0 PL=0
MOVL C00888 V=800.0 PL=0
MOVL C00889 V=800.0 PL=0
MOVL C00890 V=800.0 PL=0
MOVL C00891 V=800.0 PL=0
MOVL C00892 V=800.0 PL=0
MOVL C00893 V=800.0 PL=0
MOVL C00894 V=800.0 PL=0
MOVL C00895 V=800.0 PL=0
MOVL C00896 V=800.0 PL=0
MOVL C00897 V=800.0 PL=0
MOVL C00898 V=800.0 PL=0
MOVL C00899 V=800.0 PL=0
MOVL C00900 V=800.0 PL=0
MOVL C00901 V=800.0 PL=0
MOVL C00902 V=800.0 PL=0
MOVL C00903 V=800.0 PL=0
MOVL C00904 V=800.0 PL=0
MOVL C00905 V=800.0 PL=0
MOVL C00906 V=800.0 PL=0
MOVL C00907 V=800.0 PL=0
MOVL C00908 V=800.0 PL=0
MOVL C00909 V=800.0 PL=0
MOVL C00910 V=800.0 PL=0
MOVL C00911 V=800.0 PL=0
MOVL C00912 V=800.0 PL=0
MOVL C00913 V=800.0 PL=0
MOVL C00914 V=800.0 PL=0
MOVL C00915 V=800.0 PL=0
MOVL C00916 V=800.0 PL=0
MOVL C00917 V=800.0 PL=0
MOVL C00918 V=800.0 PL=0
MOVL C00919 V=800.0 PL=0
MOVL C00920 V=800.0 PL=0
MOVL C00921 V=800.0 PL=0
MOVL C00922 V=800.0 PL=0
MOVL C00923 V=800.0 PL=0
MOVL C00924 V=800.0 PL=0
MOVL C00925 V=800.0 PL=0
MOVL C00926 V=800.0 PL=0
MOVL C00927 V=800.0 PL=0
MOVL C00928 V=800.0 PL=0
MOVL C00929 V=800.0 PL=0
MOVL C00930 V=800.0 PL=0
MOVL C00931 V=800.0 PL=0
MOVL C00932 V=800.0 PL=0
MOVL C00933 V=800.0 PL=0
MOVL C00934 V=800.0 PL=0
MOVL C00935 V=800.0 PL=0
MOVL C00936 V=800.0 PL=0
MOVL C00937 V=800.0 PL=0
MOVL C00938 V=800.0 PL=0
MOVL C00939 V=800.0 PL=0
MOVL C00940 V=800.0 PL=0
MOVL C00941 V=800.0 PL=0
MOVL C00942 V=800.0 PL=0
MOVL C00943 V=800.0 PL=0
MOVL C00944 V=800.0 PL=0
MOVL C00945 V=800.0 PL=0
MOVL C00946 V=800.0 PL=0
MOVL C00947 V=800.0 PL=0
MOVL C00948 V=800.0 PL=0
MOVL C00949 V=800.0 PL=0
MOVL C00950 V=800.0 PL=0
MOVL C00951 V=800.0 PL=0
MOVL C00952 V=800.0 PL=0
MOVL C00953 V=800.0 PL=0
MOVL C00954 V=800.0 PL=0
MOVL C00955 V=800.0 PL=0
MOVL C00956 V=800.0 PL=0
MOVL C00957 V=800.0 PL=0
MOVL C00958 V=800.0 PL=0
MOVL C00959 V=800.0 PL=0
MOVL C00960 V=800.0 PL=0
MOVL C00961 V=800.0 PL=0
MOVL C00962 V=800.0 PL=0
MOVL C00963 V=800.0 PL=0
MOVL C00964 V=800.0 PL=0
MOVL C00965 V=800.0 PL=0
MOVL C00966 V=800.0 PL=0
MOVL C00967 V=800.0 PL=0
MOVL C00968 V=800.0 PL=0
MOVL C00969 V=800.0 PL=0
MOVL C00970 V=800.0 PL=0
MOVL C00971 V=800.0 PL=0
MOVL C00972 V=800.0 PL=0
MOVL C00973 V=800.0 PL=0
MOVL C00974 V=800.0 PL=0
MOVL C00975 V=800.0 PL=0
MOVL C00976 V=800.0 PL=0
MOVL C00977 V=800.0 PL=0
MOVL C00978 V=800.0 PL=0
MOVL C00979 V=800.0 PL=0
MOVL C00980 V=800.0 PL=0
MOVL C00981 V=800.0 PL=0
MOVL C00982 V=800.0 PL=0
MOVL C00983 V=800.0 PL=0
MOVL C00984 V=800.0 PL=0
MOVL C00985 V=800.0 PL=0
MOVL C00986 V=800.0 PL=0
MOVL C00987 V=800.0 PL=0
MOVL C00988 V=800.0 PL=0
MOVL C00989 V=800.0 PL=0
MOVL C00990 V=800.0 PL=0
MOVL C00991 V=800.0 PL=0
MOVL C00992 V=800.0 PL=0
MOVL C00993 V=800.0 PL=0
MOVL C00994 V=800.0 PL=0
MOVL C00995 V=800.0 PL=0
MOVL C00996 V=800.0 PL=0
MOVL C00997 V=800.0 PL=0
MOVL C00998 V=800.0 PL=0
MOVL C00999 V=800.0 PL=0
MOVL C01000 V=800.0 PL=0
MOVL C01001 V=800.0 PL=0
MOVL C01002 V=800.0 PL=0
MOVL C01003 V=800.0 PL=0
MOVL C01004 V=800.0 PL=0
MOVL C01005 V=800.0 PL=0
MOVL C01006 V=800.0 PL=0
MOVL C01007 V=800.0 PL=0
MOVL C01008 V=800.0 PL=0
MOVL C01009 V=800.0 PL=0
MOVL C01010 V=800.0 PL=0
MOVL C01011 V=800.0 PL=0
MOVL C01012 V=800.0 PL=0
MOVL C01013 V=800.0 PL=0
MOVL C01014 V=800.0 PL=0
MOVL C01015 V=800.0 PL=0
MOVL C01016 V=800.0 PL=0
MOVL C01017 V=800.0 PL=0
MOVL C01018 V=800.0 PL=0
MOVL C01019 V=800.0 PL=0
MOVL C01020 V=800.0 PL=0
MOVL C01021 V=800.0 PL=0
MOVL C01022 V=800.0 PL=0
MOVL C01023 V=800.0 PL=0
MOVL C01024 V=800.0 PL=0
MOVL C01025 V=800.0 PL=0
MOVL C01026 V=800.0 PL=0
MOVL C01027 V=800.0 PL=0
MOVL C01028 V=800.0 PL=0
MOVL C01029 V=800.0 PL=0
MOVL C01030 V=800.0 PL=0
MOVL C01031 V=800.0 PL=0
MOVL C01032 V=800.0 PL=0
MOVL C01033 V=800.0 PL=0
MOVL C01034 V=800.0 PL=0
MOVL C01035 V=800.0 PL=0
MOVL C01036 V=800.0 PL=0
MOVL C01037 V=800.0 PL=0
MOVL C01038 V=800.0 PL=0
MOVL C01039 V=800.0 PL=0
MOVL C01040 V=800.0 PL=0
MOVL C01041 V=800.0 PL=0
MOVL C01042 V=800.0 PL=0
MOVL C01043 V=800.0 PL=0
MOVL C01044 V=800.0 PL=0
MOVL C01045 V=800.0 PL=0
MOVL C01046 V=800.0 PL=0
MOVL C01047 V=800.0 PL=0
MOVL C01048 V=800.0 PL=0
MOVL C01049 V=800.0 PL=0
MOVL C01050 V=800.0 PL=0
MOVL C01051 V=800.0 PL=0
MOVL C01052 V=800.0 PL=0
MOVL C01053 V=800.0 PL=0
MOVL C01054 V=800.0 PL=0
MOVL C01055 V=800.0 PL=0
MOVL C01056 V=800.0 PL=0
MOVL C01057 V=800.0 PL=0
MOVL C01058 V=800.0 PL=0
MOVL C01059 V=800.0 PL=0
MOVL C01060 V=800.0 PL=0
MOVL C01061 V=800.0 PL=0
MOVL C01062 V=800.0 PL=0
MOVL C01063 V=800.0 PL=0
MOVL C01064 V=800.0 PL=0
MOVL C01065 V=800.0 PL=0
MOVL C01066 V=800.0 PL=0
MOVL C01067 V=800.0 PL=0
MOVL C01068 V=800.0 PL=0
MOVL C01069 V=800.0 PL=0
MOVL C01070 V=800.0 PL=0
MOVL C01071 V=800.0 PL=0
MOVL C01072 V=800.0 PL=0
MOVL C01073 V=800.0 PL=0
MOVL C01074 V=800.0 PL=0
MOVL C01075 V=800.0 PL=0
MOVL C01076 V=800.0 PL=0
MOVL C01077 V=800.0 PL=0
MOVL C01078 V=800.0 PL=0
MOVL C01079 V=800.0 PL=0
MOVL C01080 V=800.0 PL=0
MOVL C01081 V=800.0 PL=0
MOVL C01082 V=800.0 PL=0
MOVL C01083 V=800.0 PL=0
MOVL C01084 V=800.0 PL=0
MOVL C01085 V=800.0 PL=0
MOVL C01086 V=800.0 PL=0
MOVL C01087 V=800.0 PL=0
MOVL C01088 V=800.0 PL=0
MOVL C01089 V=800.0 PL=0
MOVL C01090 V=800.0 PL=0
MOVL C01091 V=800.0 PL=0
MOVL C01092 V=800.0 PL=0
MOVL C01093 V=800.0 PL=0
MOVL C01094 V=800.0 PL=0
MOVL C01095 V=800.0 PL=0
MOVL C01096 V=800.0 PL=0
MOVL C01097 V=800.0 PL=0
MOVL C01098 V=800.0 PL=0
MOVL C01099 V=800.0 PL=0
MOVL C01100 V=800.0 PL=0
MOVL C01101 V=800.0 PL=0
MOVL C01102 V=800.0 PL=0
MOVL C01103 V=800.0 PL=0
MOVL C01104 V=800.0 PL=0
MOVL C01105 V=800.0 PL=0
MOVL C01106 V=800.0 PL=0
MOVL C01107 V=800.0 PL=0
MOVL C01108 V=800.0 PL=0
MOVL C01109 V=800.0 PL=0
MOVL C01110 V=800.0 PL=0
MOVL C01111 V=800.0 PL=0
MOVL C01112 V=800.0 PL=0
MOVL C01113 V=800.0 PL=0
MOVL C01114 V=800.0 PL=0
MOVL C01115 V=800.0 PL=0
MOVL C01116 V=800.0 PL=0
MOVL C01117 V=800.0 PL=0
MOVL C01118 V=800.0 PL=0
MOVL C01119 V=800.0 PL=0
MOVL C01120 V=800.0 PL=0
MOVL C01121 V=800.0 PL=0
MOVL C01122 V=800.0 PL=0
MOVL C01123 V=800.0 PL=0
MOVL C01124 V=800.0 PL=0
MOVL C01125 V=800.0 PL=0
MOVL C01126 V=800.0 PL=0
MOVL C01127 V=800.0 PL=0
MOVL C01128 V=800.0 PL=0
MOVL C01129 V=800.0 PL=0
MOVL C01130 V=800.0 PL=0
MOVL C01131 V=800.0 PL=0
MOVL C01132 V=800.0 PL=0
MOVL C01133 V=800.0 PL=0
MOVL C01134 V=800.0 PL=0
MOVL C01135 V=800.0 PL=0
MOVL C01136 V=800.0 PL=0
MOVL C01137 V=800.0 PL=0
MOVL C01138 V=800.0 PL=0
MOVL C01139 V=800.0 PL=0
MOVL C01140 V=800.0 PL=0
MOVL C01141 V=800.0 PL=0
MOVL C01142 V=800.0 PL=0
MOVL C01143 V=800.0 PL=0
MOVL C01144 V=800.0 PL=0
MOVL C01145 V=800.0 PL=0
MOVL C01146 V=800.0 PL=0
MOVL C01147 V=800.0 PL=0
MOVL C01148 V=800.0 PL=0
MOVL C01149 V=800.0 PL=0
MOVL C01150 V=800.0 PL=0
MOVL C01151 V=800.0 PL=0
MOVL C01152 V=800.0 PL=0
MOVL C01153 V=800.0 PL=0
MOVL C01154 V=800.0 PL=0
MOVL C01155 V=800.0 PL=0
MOVL C01156 V=800.0 PL=0
MOVL C01157 V=800.0 PL=0
MOVL C01158 V=800.0 PL=0
MOVL C01159 V=800.0 PL=0
MOVL C01160 V=800.0 PL=0
MOVL C01161 V=800.0 PL=0
MOVL C01162 V=800.0 PL=0
MOVL C01163 V=800.0 PL=0
MOVL C01164 V=800.0 PL=0
MOVL C01165 V=800.0 PL=0
MOVL C01166 V=800.0 PL=0
MOVL C01167 V=800.0 PL=0
MOVL C01168 V=800.0 PL=0
MOVL C01169 V=800.0 PL=0
MOVL C01170 V=800.0 PL=0
MOVL C01171 V=800.0 PL=0
MOVL C01172 V=800.0 PL=0
MOVL C01173 V=800.0 PL=0
MOVL C01174 V=800.0 PL=0
MOVL C01175 V=800.0 PL=0
MOVL C01176 V=800.0 PL=0
MOVL C01177 V=800.0 PL=0
MOVL C01178 V=800.0 PL=0
MOVL C01179 V=800.0 PL=0
MOVL C01180 V=800.0 PL=0
MOVL C01181 V=800.0 PL=0
MOVL C01182 V=800.0 PL=0
MOVL C01183 V=800.0 PL=0
MOVL C01184 V=800.0 PL=0
MOVL C01185 V=800.0 PL=0
MOVL C01186 V=800.0 PL=0
MOVL C01187 V=800.0 PL=0
MOVL C01188 V=800.0 PL=0
MOVL C01189 V=800.0 PL=0
MOVL C01190 V=800.0 PL=0
MOVL C01191 V=800.0 PL=0
MOVL C01192 V=800.0 PL=0
MOVL C01193 V=800.0 PL=0
MOVL C01194 V=800.0 PL=0
MOVL C01195 V=800.0 PL=0
MOVL C01196 V=800.0 PL=0
MOVL C01197 V=800.0 PL=0
MOVL C01198 V=800.0 PL=0
MOVL C01199 V=800.0 PL=0
MOVL C01200 V=800.0 PL=0
MOVL C01201 V=800.0 PL=0
MOVL C01202 V=800.0 PL=0
MOVL C01203 V=800.0 PL=0
MOVL C01204 V=800.0 PL=0
MOVL C01205 V=800.0 PL=0
MOVL C01206 V=800.0 PL=0
MOVL C01207 V=800.0 PL=0
MOVL C01208 V=800.0 PL=0
MOVL C01209 V=800.0 PL=0
MOVL C01210 V=800.0 PL=0
MOVL C01211 V=800.0 PL=0
MOVL C01212 V=800.0 PL=0
MOVL C01213 V=800.0 PL=0
MOVL C01214 V=800.0 PL=0
MOVL C01215 V=800.0 PL=0
MOVL C01216 V=800.0 PL=0
MOVL C01217 V=800.0 PL=0
MOVL C01218 V=800.0 PL=0
MOVL C01219 V=800.0 PL=0
MOVL C01220 V=800.0 PL=0
MOVL C01221 V=800.0 PL=0
MOVL C01222 V=800.0 PL=0
MOVL C01223 V=800.0 PL=0
MOVL C01224 V=800.0 PL=0
MOVL C01225 V=800.0 PL=0
MOVL C01226 V=800.0 PL=0
MOVL C01227 V=800.0 PL=0
MOVL C01228 V=800.0 PL=0
MOVL C01229 V=800.0 PL=0
MOVL C01230 V=800.0 PL=0
MOVL C01231 V=800.0 PL=0
MOVL C01232 V=800.0 PL=0
MOVL C01233 V=800.0 PL=0
MOVL C01234 V=800.0 PL=0
MOVL C01235 V=800.0 PL=0
MOVL C01236 V=800.0 PL=0
MOVL C01237 V=800.0 PL=0
MOVL C01238 V=800.0 PL=0
MOVL C01239 V=800.0 PL=0
MOVL C01240 V=800.0 PL=0
MOVL C01241 V=800.0 PL=0
MOVL C01242 V=800.0 PL=0
MOVL C01243 V=800.0 PL=0
MOVL C01244 V=800.0 PL=0
MOVL C01245 V=800.0 PL=0
MOVL C01246 V=800.0 PL=0
MOVL C01247 V=800.0 PL=0
MOVL C01248 V=800.0 PL=0
MOVL C01249 V=800.0 PL=0
MOVL C01250 V=800.0 PL=0
MOVL C01251 V=800.0 PL=0
MOVL C01252 V=800.0 PL=0
MOVL C01253 V=800.0 PL=0
MOVL C01254 V=800.0 PL=0
MOVL C01255 V=800.0 PL=0
MOVL C01256 V=800.0 PL=0
MOVL C01257 V=800.0 PL=0
MOVL C01258 V=800.0 PL=0
MOVL C01259 V=800.0 PL=0
MOVL C01260 V=800.0 PL=0
MOVL C01261 V=800.0 PL=0
MOVL C01262 V=800.0 PL=0
MOVL C01263 V=800.0 PL=0
MOVL C01264 V=800.0 PL=0
MOVL C01265 V=800.0 PL=0
MOVL C01266 V=800.0 PL=0
MOVL C01267 V=800.0 PL=0
MOVL C01268 V=800.0 PL=0
MOVL C01269 V=800.0 PL=0
MOVL C01270 V=800.0 PL=0
MOVL C01271 V=800.0 PL=0
MOVL C01272 V=800.0 PL=0
MOVL C01273 V=800.0 PL=0
MOVL C01274 V=800.0 PL=0
MOVL C01275 V=800.0 PL=0
MOVL C01276 V=800.0 PL=0
MOVL C01277 V=800.0 PL=0
MOVL C01278 V=800.0 PL=0
MOVL C01279 V=800.0 PL=0
MOVL C01280 V=800.0 PL=0
MOVL C01281 V=800.0 PL=0
MOVL C01282 V=800.0 PL=0
MOVL C01283 V=800.0 PL=0
MOVL C01284 V=800.0 PL=0
MOVL C01285 V=800.0 PL=0
MOVL C01286 V=800.0 PL=0
MOVL C01287 V=800.0 PL=0
MOVL C01288 V=800.0 PL=0
MOVL C01289 V=800.0 PL=0
MOVL C01290 V=800.0 PL=0
MOVL C01291 V=800.0 PL=0
MOVL C01292 V=800.0 PL=0
MOVL C01293 V=800.0 PL=0
MOVL C01294 V=800.0 PL=0
MOVL C01295 V=800.0 PL=0
MOVL C01296 V=800.0 PL=0
MOVL C01297 V=800.0 PL=0
MOVL C01298 V=800.0 PL=0
MOVL C01299 V=800.0 PL=0
MOVL C01300 V=800.0 PL=0
MOVL C01301 V=800.0 PL=0
MOVL C01302 V=800.0 PL=0
MOVL C01303 V=800.0 PL=0
MOVL C01304 V=800.0 PL=0
MOVL C01305 V=800.0 PL=0
MOVL C01306 V=800.0 PL=0
MOVL C01307 V=800.0 PL=0
MOVL C01308 V=800.0 PL=0
MOVL C01309 V=800.0 PL=0
MOVL C01310 V=800.0 PL=0
MOVL C01311 V=800.0 PL=0
MOVL C01312 V=800.0 PL=0
MOVL C01313 V=800.0 PL=0
MOVL C01314 V=800.0 PL=0
MOVL C01315 V=800.0 PL=0
MOVL C01316 V=800.0 PL=0
MOVL C01317 V=800.0 PL=0
MOVL C01318 V=800.0 PL=0
MOVL C01319 V=800.0 PL=0
MOVL C01320 V=800.0 PL=0
MOVL C01321 V=800.0 PL=0
MOVL C01322 V=800.0 PL=0
MOVL C01323 V=800.0 PL=0
MOVL C01324 V=800.0 PL=0
MOVL C01325 V=800.0 PL=0
MOVL C01326 V=800.0 PL=0
MOVL C01327 V=800.0 PL=0
MOVL C01328 V=800.0 PL=0
MOVL C01329 V=800.0 PL=0
MOVL C01330 V=800.0 PL=0
MOVL C01331 V=800.0 PL=0
MOVL C01332 V=800.0 PL=0
MOVL C01333 V=800.0 PL=0
MOVL C01334 V=800.0 PL=0
MOVL C01335 V=800.0 PL=0
MOVL C01336 V=800.0 PL=0
MOVL C01337 V=800.0 PL=0
MOVL C01338 V=800.0 PL=0
MOVL C01339 V=800.0 PL=0
MOVL C01340 V=800.0 PL=0
MOVL C01341 V=800.0 PL=0
MOVL C01342 V=800.0 PL=0
MOVL C01343 V=800.0 PL=0
MOVL C01344 V=800.0 PL=0
MOVL C01345 V=800.0 PL=0
MOVL C01346 V=800.0 PL=0
MOVL C01347 V=800.0 PL=0
MOVL C01348 V=800.0 PL=0
MOVL C01349 V=800.0 PL=0
MOVL C01350 V=800.0 PL=0
MOVL C01351 V=800.0 PL=0
MOVL C01352 V=800.0 PL=0
MOVL C01353 V=800.0 PL=0
MOVL C01354 V=800.0 PL=0
MOVL C01355 V=800.0 PL=0
MOVL C01356 V=800.0 PL=0
MOVL C01357 V=800.0 PL=0
MOVL C01358 V=800.0 PL=0
MOVL C01359 V=800.0 PL=0
MOVL C01360 V=800.0 PL=0
MOVL C01361 V=800.0 PL=0
MOVL C01362 V=800.0 PL=0
MOVL C01363 V=800.0 PL=0
MOVL C01364 V=800.0 PL=0
MOVL C01365 V=800.0 PL=0
MOVL C01366 V=800.0 PL=0
MOVL C01367 V=800.0 PL=0
MOVL C01368 V=800.0 PL=0
MOVL C01369 V=800.0 PL=0
MOVL C01370 V=800.0 PL=0
MOVL C01371 V=800.0 PL=0
MOVL C01372 V=800.0 PL=0
MOVL C01373 V=800.0 PL=0
MOVL C01374 V=800.0 PL=0
MOVL C01375 V=800.0 PL=0
MOVL C01376 V=800.0 PL=0
MOVL C01377 V=800.0 PL=0
MOVL C01378 V=800.0 PL=0
MOVL C01379 V=800.0 PL=0
MOVL C01380 V=800.0 PL=0
MOVL C01381 V=800.0 PL=0
MOVL C01382 V=800.0 PL=0
MOVL C01383 V=800.0 PL=0
MOVL C01384 V=800.0 PL=0
MOVL C01385 V=800.0 PL=0
MOVL C01386 V=800.0 PL=0
MOVL C01387 V=800.0 PL=0
MOVL C01388 V=800.0 PL=0
MOVL C01389 V=800.0 PL=0
MOVL C01390 V=800.0 PL=0
MOVL C01391 V=800.0 PL=0
MOVL C01392 V=800.0 PL=0
MOVL C01393 V=800.0 PL=0
MOVL C01394 V=800.0 PL=0
MOVL C01395 V=800.0 PL=0
MOVL C01396 V=800.0 PL=0
MOVL C01397 V=800.0 PL=0
MOVL C01398 V=800.0 PL=0
MOVL C01399 V=800.0 PL=0
MOVL C01400 V=800.0 PL=0
MOVL C01401 V=800.0 PL=0
MOVL C01402 V=800.0 PL=0
MOVL C01403 V=800.0 PL=0
MOVL C01404 V=800.0 PL=0
MOVL C01405 V=800.0 PL=0
MOVL C01406 V=800.0 PL=0
MOVL C01407 V=800.0 PL=0
MOVL C01408 V=800.0 PL=0
MOVL C01409 V=800.0 PL=0
MOVL C01410 V=800.0 PL=0
MOVL C01411 V=800.0 PL=0
MOVL C01412 V=800.0 PL=0
MOVL C01413 V=800.0 PL=0
MOVL C01414 V=800.0 PL=0
MOVL C01415 V=800.0 PL=0
MOVL C01416 V=800.0 PL=0
MOVL C01417 V=800.0 PL=0
MOVL C01418 V=800.0 PL=0
MOVL C01419 V=800.0 PL=0
MOVL C01420 V=800.0 PL=0
MOVL C01421 V=800.0 PL=0
MOVL C01422 V=800.0 PL=0
MOVL C01423 V=800.0 PL=0
MOVL C01424 V=800.0 PL=0
MOVL C01425 V=800.0 PL=0
MOVL C01426 V=800.0 PL=0
MOVL C01427 V=800.0 PL=0
MOVL C01428 V=800.0 PL=0
MOVL C01429 V=800.0 PL=0
MOVL C01430 V=800.0 PL=0
MOVL C01431 V=800.0 PL=0
MOVL C01432 V=800.0 PL=0
MOVL C01433 V=800.0 PL=0
MOVL C01434 V=800.0 PL=0
MOVL C01435 V=800.0 PL=0
MOVL C01436 V=800.0 PL=0
MOVL C01437 V=800.0 PL=0
MOVL C01438 V=800.0 PL=0
MOVL C01439 V=800.0 PL=0
MOVL C01440 V=800.0 PL=0
MOVL C01441 V=800.0 PL=0
MOVL C01442 V=800.0 PL=0
MOVL C01443 V=800.0 PL=0
MOVL C01444 V=800.0 PL=0
MOVL C01445 V=800.0 PL=0
MOVL C01446 V=800.0 PL=0
MOVL C01447 V=800.0 PL=0
MOVL C01448 V=800.0 PL=0
MOVL C01449 V=800.0 PL=0
MOVL C01450 V=800.0 PL=0
MOVL C01451 V=800.0 PL=0
MOVL C01452 V=800.0 PL=0
MOVL C01453 V=800.0 PL=0
MOVL C01454 V=800.0 PL=0
MOVL C01455 V=800.0 PL=0
MOVL C01456 V=800.0 PL=0
MOVL C01457 V=800.0 PL=0
MOVL C01458 V=800.0 PL=0
MOVL C01459 V=800.0 PL=0
MOVL C01460 V=800.0 PL=0
MOVL C01461 V=800.0 PL=0
MOVL C01462 V=800.0 PL=0
MOVL C01463 V=800.0 PL=0
MOVL C01464 V=800.0 PL=0
MOVL C01465 V=800.0 PL=0
MOVL C01466 V=800.0 PL=0
MOVL C01467 V=800.0 PL=0
MOVL C01468 V=800.0 PL=0
MOVL C01469 V=800.0 PL=0
MOVL C01470 V=800.0 PL=0
MOVL C01471 V=800.0 PL=0
MOVL C01472 V=800.0 PL=0
MOVL C01473 V=800.0 PL=0
MOVL C01474 V=800.0 PL=0
MOVL C01475 V=800.0 PL=0
MOVL C01476 V=800.0 PL=0
MOVL C01477 V=800.0 PL=0
MOVL C01478 V=800.0 PL=0
MOVL C01479 V=800.0 PL=0
MOVL C01480 V=800.0 PL=0
MOVL C01481 V=800.0 PL=0
MOVL C01482 V=800.0 PL=0
MOVL C01483 V=800.0 PL=0
MOVL C01484 V=800.0 PL=0
MOVL C01485 V=800.0 PL=0
MOVL C01486 V=800.0 PL=0
MOVL C01487 V=800.0 PL=0
MOVL C01488 V=800.0 PL=0
MOVL C01489 V=800.0 PL=0
MOVL C01490 V=800.0 PL=0
MOVL C01491 V=800.0 PL=0
MOVL C01492 V=800.0 PL=0
MOVL C01493 V=800.0 PL=0
MOVL C01494 V=800.0 PL=0
MOVL C01495 V=800.0 PL=0
MOVL C01496 V=800.0 PL=0
MOVL C01497 V=800.0 PL=0
MOVL C01498 V=800.0 PL=0
MOVL C01499 V=800.0 PL=0
MOVL C01500 V=800.0 PL=0
MOVL C01501 V=800.0 PL=0
MOVL C01502 V=800.0 PL=0
MOVL C01503 V=800.0 PL=0
MOVL C01504 V=800.0 PL=0
MOVL C01505 V=800.0 PL=0
MOVL C01506 V=800.0 PL=0
MOVL C01507 V=800.0 PL=0
MOVL C01508 V=800.0 PL=0
MOVL C01509 V=800.0 PL=0
MOVL C01510 V=800.0 PL=0
MOVL C01511 V=800.0 PL=0
MOVL C01512 V=800.0 PL=0
MOVL C01513 V=800.0 PL=0
MOVL C01514 V=800.0 PL=0
MOVL C01515 V=800.0 PL=0
MOVL C01516 V=800.0 PL=0
MOVL C01517 V=800.0 PL=0
MOVL C01518 V=800.0 PL=0
MOVL C01519 V=800.0 PL=0
MOVL C01520 V=800.0 PL=0
MOVL C01521 V=800.0 PL=0
MOVL C01522 V=800.0 PL=0
MOVL C01523 V=800.0 PL=0
MOVL C01524 V=800.0 PL=0
MOVL C01525 V=800.0 PL=0
MOVL C01526 V=800.0 PL=0
MOVL C01527 V=800.0 PL=0
MOVL C01528 V=800.0 PL=0
MOVL C01529 V=800.0 PL=0
MOVL C01530 V=800.0 PL=0
MOVL C01531 V=800.0 PL=0
MOVL C01532 V=800.0 PL=0
MOVL C01533 V=800.0 PL=0
MOVL C01534 V=800.0 PL=0
MOVL C01535 V=800.0 PL=0
MOVL C01536 V=800.0 PL=0
MOVL C01537 V=800.0 PL=0
MOVL C01538 V=800.0 PL=0
MOVL C01539 V=800.0 PL=0
MOVL C01540 V=800.0 PL=0
MOVL C01541 V=800.0 PL=0
MOVL C01542 V=800.0 PL=0
MOVL C01543 V=800.0 PL=0
MOVL C01544 V=800.0 PL=0
MOVL C01545 V=800.0 PL=0
MOVL C01546 V=800.0 PL=0
MOVL C01547 V=800.0 PL=0
MOVL C01548 V=800.0 PL=0
MOVL C01549 V=800.0 PL=0
MOVL C01550 V=800.0 PL=0
MOVL C01551 V=800.0 PL=0
MOVL C01552 V=800.0 PL=0
MOVL C01553 V=800.0 PL=0
MOVL C01554 V=800.0 PL=0
MOVL C01555 V=800.0 PL=0
MOVL C01556 V=800.0 PL=0
MOVL C01557 V=800.0 PL=0
MOVL C01558 V=800.0 PL=0
MOVL C01559 V=800.0 PL=0
MOVL C01560 V=800.0 PL=0
MOVL C01561 V=800.0 PL=0
MOVL C01562 V=800.0 PL=0
MOVL C01563 V=800.0 PL=0
MOVL C01564 V=800.0 PL=0
MOVL C01565 V=800.0 PL=0
MOVL C01566 V=800.0 PL=0
MOVL C01567 V=800.0 PL=0
MOVL C01568 V=800.0 PL=0
MOVL C01569 V=800.0 PL=0
MOVL C01570 V=800.0 PL=0
MOVL C01571 V=800.0 PL=0
MOVL C01572 V=800.0 PL=0
MOVL C01573 V=800.0 PL=0
MOVL C01574 V=800.0 PL=0
MOVL C01575 V=800.0 PL=0
MOVL C01576 V=800.0 PL=0
MOVL C01577 V=800.0 PL=0
MOVL C01578 V=800.0 PL=0
MOVL C01579 V=800.0 PL=0
MOVL C01580 V=800.0 PL=0
MOVL C01581 V=800.0 PL=0
MOVL C01582 V=800.0 PL=0
MOVL C01583 V=800.0 PL=0
MOVL C01584 V=800.0 PL=0
MOVL C01585 V=800.0 PL=0
MOVL C01586 V=800.0 PL=0
MOVL C01587 V=800.0 PL=0
MOVL C01588 V=800.0 PL=0
MOVL C01589 V=800.0 PL=0
MOVL C01590 V=800.0 PL=0
MOVL C01591 V=800.0 PL=0
MOVL C01592 V=800.0 PL=0
MOVL C01593 V=800.0 PL=0
MOVL C01594 V=800.0 PL=0
MOVL C01595 V=800.0 PL=0
MOVL C01596 V=800.0 PL=0
MOVL C01597 V=800.0 PL=0
MOVL C01598 V=800.0 PL=0
MOVL C01599 V=800.0 PL=0
MOVL C01600 V=800.0 PL=0
MOVL C01601 V=800.0 PL=0
MOVL C01602 V=800.0 PL=0
MOVL C01603 V=800.0 PL=0
MOVL C01604 V=800.0 PL=0
MOVL C01605 V=800.0 PL=0
MOVL C01606 V=800.0 PL=0
MOVL C01607 V=800.0 PL=0
MOVL C01608 V=800.0 PL=0
MOVL C01609 V=800.0 PL=0
MOVL C01610 V=800.0 PL=0
MOVL C01611 V=800.0 PL=0
MOVL C01612 V=800.0 PL=0
MOVL C01613 V=800.0 PL=0
MOVL C01614 V=800.0 PL=0
MOVL C01615 V=800.0 PL=0
MOVL C01616 V=800.0 PL=0
MOVL C01617 V=800.0 PL=0
MOVL C01618 V=800.0 PL=0
MOVL C01619 V=800.0 PL=0
MOVL C01620 V=800.0 PL=0
MOVL C01621 V=800.0 PL=0
MOVL C01622 V=800.0 PL=0
MOVL C01623 V=800.0 PL=0
MOVL C01624 V=800.0 PL=0
MOVL C01625 V=800.0 PL=0
MOVL C01626 V=800.0 PL=0
MOVL C01627 V=800.0 PL=0
MOVL C01628 V=800.0 PL=0
MOVL C01629 V=800.0 PL=0
MOVL C01630 V=800.0 PL=0
MOVL C01631 V=800.0 PL=0
MOVL C01632 V=800.0 PL=0
MOVL C01633 V=800.0 PL=0
MOVL C01634 V=800.0 PL=0
MOVL C01635 V=800.0 PL=0
MOVL C01636 V=800.0 PL=0
MOVL C01637 V=800.0 PL=0
MOVL C01638 V=800.0 PL=0
MOVL C01639 V=800.0 PL=0
MOVL C01640 V=800.0 PL=0
MOVL C01641 V=800.0 PL=0
MOVL C01642 V=800.0 PL=0
MOVL C01643 V=800.0 PL=0
MOVL C01644 V=800.0 PL=0
MOVL C01645 V=800.0 PL=0
MOVL C01646 V=800.0 PL=0
MOVL C01647 V=800.0 PL=0
MOVL C01648 V=800.0 PL=0
MOVL C01649 V=800.0 PL=0
MOVL C01650 V=800.0 PL=0
MOVL C01651 V=800.0 PL=0
MOVL C01652 V=800.0 PL=0
MOVL C01653 V=800.0 PL=0
MOVL C01654 V=800.0 PL=0
MOVL C01655 V=800.0 PL=0
MOVL C01656 V=800.0 PL=0
MOVL C01657 V=800.0 PL=0
MOVL C01658 V=800.0 PL=0
MOVL C01659 V=800.0 PL=0
MOVL C01660 V=800.0 PL=0
MOVL C01661 V=800.0 PL=0
MOVL C01662 V=800.0 PL=0
MOVL C01663 V=800.0 PL=0
MOVL C01664 V=800.0 PL=0
MOVL C01665 V=800.0 PL=0
MOVL C01666 V=800.0 PL=0
MOVL C01667 V=800.0 PL=0
MOVL C01668 V=800.0 PL=0
MOVL C01669 V=800.0 PL=0
MOVL C01670 V=800.0 PL=0
MOVL C01671 V=800.0 PL=0
MOVL C01672 V=800.0 PL=0
MOVL C01673 V=800.0 PL=0
MOVL C01674 V=800.0 PL=0
MOVL C01675 V=800.0 PL=0
MOVL C01676 V=800.0 PL=0
MOVL C01677 V=800.0 PL=0
MOVL C01678 V=800.0 PL=0
MOVL C01679 V=800.0 PL=0
MOVL C01680 V=800.0 PL=0
MOVL C01681 V=800.0 PL=0
MOVL C01682 V=800.0 PL=0
MOVL C01683 V=800.0 PL=0
MOVL C01684 V=800.0 PL=0
MOVL C01685 V=800.0 PL=0
MOVL C01686 V=800.0 PL=0
MOVL C01687 V=800.0 PL=0
MOVL C01688 V=800.0 PL=0
MOVL C01689 V=800.0 PL=0
MOVL C01690 V=800.0 PL=0
MOVL C01691 V=800.0 PL=0
MOVL C01692 V=800.0 PL=0
MOVL C01693 V=800.0 PL=0
MOVL C01694 V=800.0 PL=0
MOVL C01695 V=800.0 PL=0
MOVL C01696 V=800.0 PL=0
MOVL C01697 V=800.0 PL=0
MOVL C01698 V=800.0 PL=0
MOVL C01699 V=800.0 PL=0
MOVL C01700 V=800.0 PL=0
MOVL C01701 V=800.0 PL=0
MOVL C01702 V=800.0 PL=0
MOVL C01703 V=800.0 PL=0
MOVL C01704 V=800.0 PL=0
MOVL C01705 V=800.0 PL=0
MOVL C01706 V=800.0 PL=0
MOVL C01707 V=800.0 PL=0
MOVL C01708 V=800.0 PL=0
MOVL C01709 V=800.0 PL=0
MOVL C01710 V=800.0 PL=0
MOVL C01711 V=800.0 PL=0
MOVL C01712 V=800.0 PL=0
MOVL C01713 V=800.0 PL=0
MOVL C01714 V=800.0 PL=0
MOVL C01715 V=800.0 PL=0
MOVL C01716 V=800.0 PL=0
MOVL C01717 V=800.0 PL=0
MOVL C01718 V=800.0 PL=0
MOVL C01719 V=800.0 PL=0
MOVL C01720 V=800.0 PL=0
MOVL C01721 V=800.0 PL=0
MOVL C01722 V=800.0 PL=0
MOVL C01723 V=800.0 PL=0
MOVL C01724 V=800.0 PL=0
MOVL C01725 V=800.0 PL=0
MOVL C01726 V=800.0 PL=0
MOVL C01727 V=800.0 PL=0
MOVL C01728 V=800.0 PL=0
MOVL C01729 V=800.0 PL=0
MOVL C01730 V=800.0 PL=0
MOVL C01731 V=800.0 PL=0
MOVL C01732 V=800.0 PL=0
MOVL C01733 V=800.0 PL=0
MOVL C01734 V=800.0 PL=0
MOVL C01735 V=800.0 PL=0
MOVL C01736 V=800.0 PL=0
MOVL C01737 V=800.0 PL=0
MOVL C01738 V=800.0 PL=0
MOVL C01739 V=800.0 PL=0
MOVL C01740 V=800.0 PL=0
MOVL C01741 V=800.0 PL=0
MOVL C01742 V=800.0 PL=0
MOVL C01743 V=800.0 PL=0
MOVL C01744 V=800.0 PL=0
MOVL C01745 V=800.0 PL=0
MOVL C01746 V=800.0 PL=0
MOVL C01747 V=800.0 PL=0
MOVL C01748 V=800.0 PL=0
MOVL C01749 V=800.0 PL=0
MOVL C01750 V=800.0 PL=0
MOVL C01751 V=800.0 PL=0
MOVL C01752 V=800.0 PL=0
MOVL C01753 V=800.0 PL=0
MOVL C01754 V=800.0 PL=0
MOVL C01755 V=800.0 PL=0
MOVL C01756 V=800.0 PL=0
MOVL C01757 V=800.0 PL=0
MOVL C01758 V=800.0 PL=0
MOVL C01759 V=800.0 PL=0
MOVL C01760 V=800.0 PL=0
MOVL C01761 V=800.0 PL=0
MOVL C01762 V=800.0 PL=0
MOVL C01763 V=800.0 PL=0
MOVL C01764 V=800.0 PL=0
MOVL C01765 V=800.0 PL=0
MOVL C01766 V=800.0 PL=0
MOVL C01767 V=800.0 PL=0
MOVL C01768 V=800.0 PL=0
MOVL C01769 V=800.0 PL=0
MOVL C01770 V=800.0 PL=0
MOVL C01771 V=800.0 PL=0
MOVL C01772 V=800.0 PL=0
MOVL C01773 V=800.0 PL=0
MOVL C01774 V=800.0 PL=0
MOVL C01775 V=800.0 PL=0
MOVL C01776 V=800.0 PL=0
MOVL C01777 V=800.0 PL=0
MOVL C01778 V=800.0 PL=0
MOVL C01779 V=800.0 PL=0
MOVL C01780 V=800.0 PL=0
MOVL C01781 V=800.0 PL=0
MOVL C01782 V=800.0 PL=0
MOVL C01783 V=800.0 PL=0
MOVL C01784 V=800.0 PL=0
MOVL C01785 V=800.0 PL=0
MOVL C01786 V=800.0 PL=0
MOVL C01787 V=800.0 PL=0
MOVL C01788 V=800.0 PL=0
MOVL C01789 V=800.0 PL=0
MOVL C01790 V=800.0 PL=0
MOVL C01791 V=800.0 PL=0
MOVL C01792 V=800.0 PL=0
MOVL C01793 V=800.0 PL=0
MOVL C01794 V=800.0 PL=0
MOVL C01795 V=800.0 PL=0
MOVL C01796 V=800.0 PL=0
MOVL C01797 V=800.0 PL=0
MOVL C01798 V=800.0 PL=0
MOVL C01799 V=800.0 PL=0
MOVL C01800 V=800.0 PL=0
MOVL C01801 V=800.0 PL=0
MOVL C01802 V=800.0 PL=0
MOVL C01803 V=800.0 PL=0
MOVL C01804 V=800.0 PL=0
MOVL C01805 V=800.0 PL=0
MOVL C01806 V=800.0 PL=0
MOVL C01807 V=800.0 PL=0
MOVL C01808 V=800.0 PL=0
MOVL C01809 V=800.0 PL=0
MOVL C01810 V=800.0 PL=0
MOVL C01811 V=800.0 PL=0
MOVL C01812 V=800.0 PL=0
MOVL C01813 V=800.0 PL=0
MOVL C01814 V=800.0 PL=0
MOVL C01815 V=800.0 PL=0
MOVL C01816 V=800.0 PL=0
MOVL C01817 V=800.0 PL=0
MOVL C01818 V=800.0 PL=0
MOVL C01819 V=800.0 PL=0
MOVL C01820 V=800.0 PL=0
MOVL C01821 V=800.0 PL=0
MOVL C01822 V=800.0 PL=0
MOVL C01823 V=800.0 PL=0
MOVL C01824 V=800.0 PL=0
MOVL C01825 V=800.0 PL=0
MOVL C01826 V=800.0 PL=0
MOVL C01827 V=800.0 PL=0
MOVL C01828 V=800.0 PL=0
MOVL C01829 V=800.0 PL=0
MOVL C01830 V=800.0 PL=0
MOVL C01831 V=800.0 PL=0
MOVL C01832 V=800.0 PL=0
MOVL C01833 V=800.0 PL=0
MOVL C01834 V=800.0 PL=0
MOVL C01835 V=800.0 PL=0
MOVL C01836 V=800.0 PL=0
MOVL C01837 V=800.0 PL=0
MOVL C01838 V=800.0 PL=0
MOVL C01839 V=800.0 PL=0
MOVL C01840 V=800.0 PL=0
MOVL C01841 V=800.0 PL=0
MOVL C01842 V=800.0 PL=0
MOVL C01843 V=800.0 PL=0
MOVL C01844 V=800.0 PL=0
MOVL C01845 V=800.0 PL=0
MOVL C01846 V=800.0 PL=0
MOVL C01847 V=800.0 PL=0
MOVL C01848 V=800.0 PL=0
MOVL C01849 V=800.0 PL=0
MOVL C01850 V=800.0 PL=0
MOVL C01851 V=800.0 PL=0
MOVL C01852 V=800.0 PL=0
MOVL C01853 V=800.0 PL=0
MOVL C01854 V=800.0 PL=0
MOVL C01855 V=800.0 PL=0
MOVL C01856 V=800.0 PL=0
MOVL C01857 V=800.0 PL=0
MOVL C01858 V=800.0 PL=0
MOVL C01859 V=800.0 PL=0
MOVL C01860 V=800.0 PL=0
MOVL C01861 V=800.0 PL=0
MOVL C01862 V=800.0 PL=0
MOVL C01863 V=800.0 PL=0
MOVL C01864 V=800.0 PL=0
MOVL C01865 V=800.0 PL=0
MOVL C01866 V=800.0 PL=0
MOVL C01867 V=800.0 PL=0
MOVL C01868 V=800.0 PL=0
MOVL C01869 V=800.0 PL=0
MOVL C01870 V=800.0 PL=0
MOVL C01871 V=800.0 PL=0
MOVL C01872 V=800.0 PL=0
MOVL C01873 V=800.0 PL=0
MOVL C01874 V=800.0 PL=0
MOVL C01875 V=800.0 PL=0
MOVL C01876 V=800.0 PL=0
MOVL C01877 V=800.0 PL=0
MOVL C01878 V=800.0 PL=0
MOVL C01879 V=800.0 PL=0
MOVL C01880 V=800.0 PL=0
MOVL C01881 V=800.0 PL=0
MOVL C01882 V=800.0 PL=0
MOVL C01883 V=800.0 PL=0
MOVL C01884 V=800.0 PL=0
MOVL C01885 V=800.0 PL=0
MOVL C01886 V=800.0 PL=0
MOVL C01887 V=800.0 PL=0
MOVL C01888 V=800.0 PL=0
MOVL C01889 V=800.0 PL=0
MOVL C01890 V=800.0 PL=0
MOVL C01891 V=800.0 PL=0
MOVL C01892 V=800.0 PL=0
MOVL C01893 V=800.0 PL=0
MOVL C01894 V=800.0 PL=0
MOVL C01895 V=800.0 PL=0
MOVL C01896 V=800.0 PL=0
MOVL C01897 V=800.0 PL=0
MOVL C01898 V=800.0 PL=0
MOVL C01899 V=800.0 PL=0
MOVL C01900 V=800.0 PL=0
MOVL C01901 V=800.0 PL=0
MOVL C01902 V=800.0 PL=0
MOVL C01903 V=800.0 PL=0
MOVL C01904 V=800.0 PL=0
MOVL C01905 V=800.0 PL=0
MOVL C01906 V=800.0 PL=0
MOVL C01907 V=800.0 PL=0
MOVL C01908 V=800.0 PL=0
MOVL C01909 V=800.0 PL=0
MOVL C01910 V=800.0 PL=0
MOVL C01911 V=800.0 PL=0
MOVL C01912 V=800.0 PL=0
MOVL C01913 V=800.0 PL=0
MOVL C01914 V=800.0 PL=0
MOVL C01915 V=800.0 PL=0
MOVL C01916 V=800.0 PL=0
MOVL C01917 V=800.0 PL=0
MOVL C01918 V=800.0 PL=0
MOVL C01919 V=800.0 PL=0
MOVL C01920 V=800.0 PL=0
MOVL C01921 V=800.0 PL=0
MOVL C01922 V=800.0 PL=0
MOVL C01923 V=800.0 PL=0
MOVL C01924 V=800.0 PL=0
MOVL C01925 V=800.0 PL=0
MOVL C01926 V=800.0 PL=0
MOVL C01927 V=800.0 PL=0
MOVL C01928 V=800.0 PL=0
MOVL C01929 V=800.0 PL=0
MOVL C01930 V=800.0 PL=0
MOVL C01931 V=800.0 PL=0
MOVL C01932 V=800.0 PL=0
MOVL C01933 V=800.0 PL=0
MOVL C01934 V=800.0 PL=0
MOVL C01935 V=800.0 PL=0
MOVL C01936 V=800.0 PL=0
MOVL C01937 V=800.0 PL=0
MOVL C01938 V=800.0 PL=0
MOVL C01939 V=800.0 PL=0
MOVL C01940 V=800.0 PL=0
MOVL C01941 V=800.0 PL=0
MOVL C01942 V=800.0 PL=0
MOVL C01943 V=800.0 PL=0
MOVL C01944 V=800.0 PL=0
MOVL C01945 V=800.0 PL=0
MOVL C01946 V=800.0 PL=0
MOVL C01947 V=800.0 PL=0
MOVL C01948 V=800.0 PL=0
MOVL C01949 V=800.0 PL=0
MOVL C01950 V=800.0 PL=0
MOVL C01951 V=800.0 PL=0
MOVL C01952 V=800.0 PL=0
MOVL C01953 V=800.0 PL=0
MOVL C01954 V=800.0 PL=0
MOVL C01955 V=800.0 PL=0
MOVL C01956 V=800.0 PL=0
MOVL C01957 V=800.0 PL=0
MOVL C01958 V=800.0 PL=0
MOVL C01959 V=800.0 PL=0
MOVL C01960 V=800.0 PL=0
MOVL C01961 V=800.0 PL=0
MOVL C01962 V=800.0 PL=0
MOVL C01963 V=800.0 PL=0
MOVL C01964 V=800.0 PL=0
MOVL C01965 V=800.0 PL=0
MOVL C01966 V=800.0 PL=0
MOVL C01967 V=800.0 PL=0
MOVL C01968 V=800.0 PL=0
MOVL C01969 V=800.0 PL=0
MOVL C01970 V=800.0 PL=0
MOVL C01971 V=800.0 PL=0
MOVL C01972 V=800.0 PL=0
MOVL C01973 V=800.0 PL=0
MOVL C01974 V=800.0 PL=0
MOVL C01975 V=800.0 PL=0
MOVL C01976 V=800.0 PL=0
MOVL C01977 V=800.0 PL=0
MOVL C01978 V=800.0 PL=0
MOVL C01979 V=800.0 PL=0
MOVL C01980 V=800.0 PL=0
MOVL C01981 V=800.0 PL=0
MOVL C01982 V=800.0 PL=0
MOVL C01983 V=800.0 PL=0
MOVL C01984 V=800.0 PL=0
MOVL C01985 V=800.0 PL=0
MOVL C01986 V=800.0 PL=0
MOVL C01987 V=800.0 PL=0
MOVL C01988 V=800.0 PL=0
MOVL C01989 V=800.0 PL=0
MOVL C01990 V=800.0 PL=0
MOVL C01991 V=800.0 PL=0
MOVL C01992 V=800.0 PL=0
MOVL C01993 V=800.0 PL=0
MOVL C01994 V=800.0 PL=0
MOVL C01995 V=800.0 PL=0
MOVL C01996 V=800.0 PL=0
MOVL C01997 V=800.0 PL=0
MOVL C01998 V=800.0 PL=0
MOVL C01999 V=800.0 PL=0
MOVL C02000 V=800.0 PL=0
MOVL C02001 V=800.0 PL=0
MOVL C02002 V=800.0 PL=0
MOVL C02003 V=800.0 PL=0
MOVL C02004 V=800.0 PL=0
MOVL C02005 V=800.0 PL=0
MOVL C02006 V=800.0 PL=0
MOVL C02007 V=800.0 PL=0
MOVL C02008 V=800.0 PL=0
MOVL C02009 V=800.0 PL=0
MOVL C02010 V=800.0 PL=0
MOVL C02011 V=800.0 PL=0
MOVL C02012 V=800.0 PL=0
MOVL C02013 V=800.0 PL=0
MOVL C02014 V=800.0 PL=0
MOVL C02015 V=800.0 PL=0
MOVL C02016 V=800.0 PL=0
MOVL C02017 V=800.0 PL=0
MOVL C02018 V=800.0 PL=0
MOVL C02019 V=800.0 PL=0
MOVL C02020 V=800.0 PL=0
MOVL C02021 V=800.0 PL=0
MOVL C02022 V=800.0 PL=0
MOVL C02023 V=800.0 PL=0
MOVL C02024 V=800.0 PL=0
MOVL C02025 V=800.0 PL=0
MOVL C02026 V=800.0 PL=0
MOVL C02027 V=800.0 PL=0
MOVL C02028 V=800.0 PL=0
MOVL C02029 V=800.0 PL=0
MOVL C02030 V=800.0 PL=0
